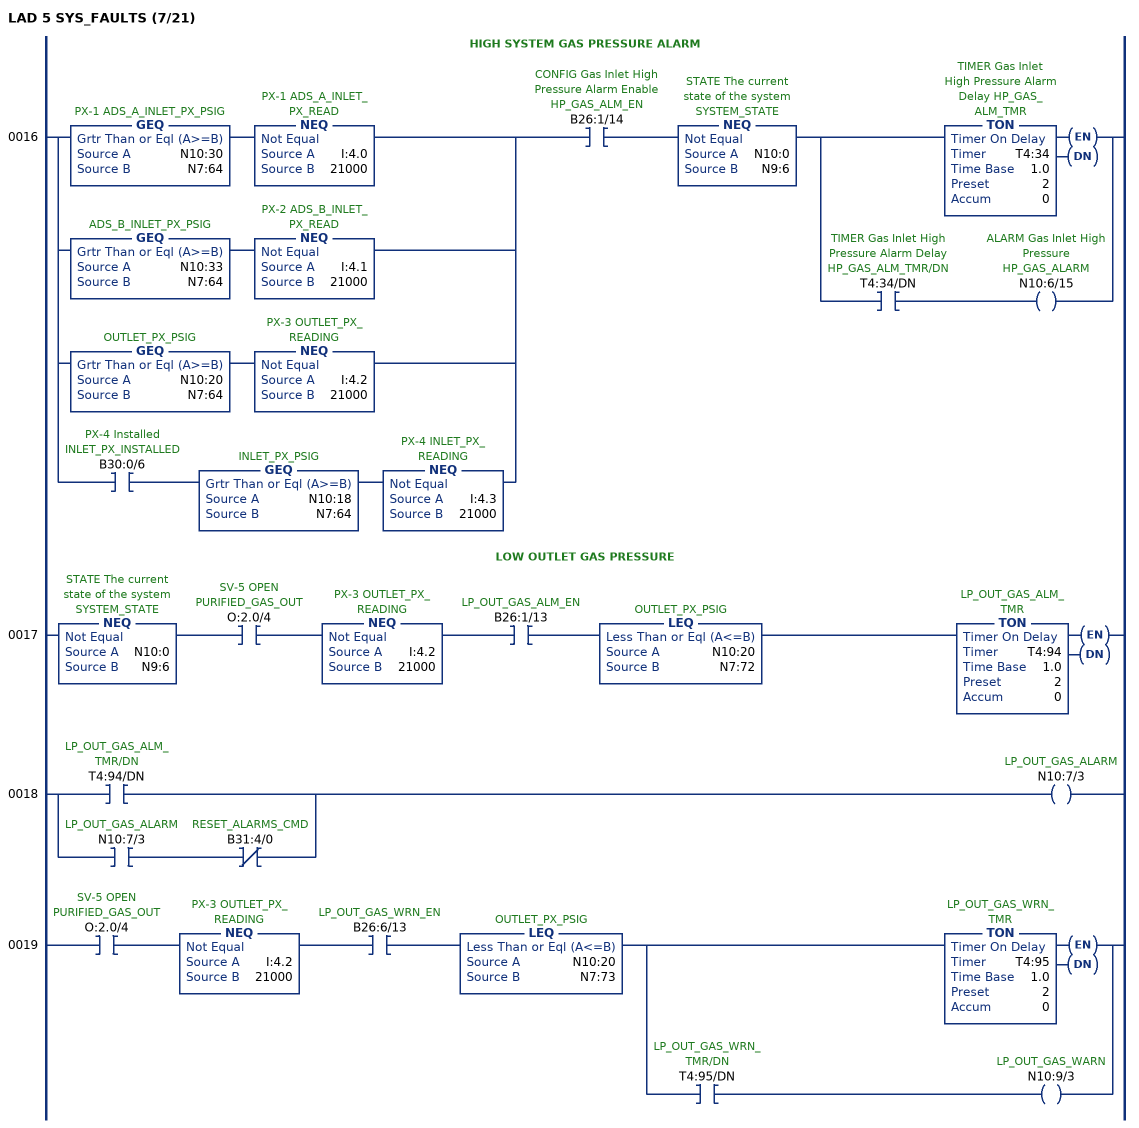
% Rung: 16 %
% TITLE: HIGH SYSTEM GAS PRESSURE ALARM %
SOR BST GEQ N10:30 N7:64 NEQ I:4.0 21000 NXB GEQ N10:33 N7:64 NEQ I:4.1 21000 NXB GEQ N10:20 N7:64 NEQ I:4.2 21000 NXB XIC B30:0/6 GEQ N10:18 N7:64 NEQ I:4.3 21000 BND XIC B26:1/14 NEQ N10:0 N9:6 BST TON T4:34 1.0 2 0 NXB XIC T4:34/DN OTE N10:6/15 BND EOR
%   N10:30  ADS_A_INLET_PX_PSIG  "PX-1" %
%   N7:64  HP_GAS_ALM_SP  "CONFIG Gas Inlet High Pressure Alarm Setpoint" %
%   I:4.0  ADS_A_INLET_PX_READ  "PX-1" %
%   N10:33  ADS_B_INLET_PX_PSIG %
%   I:4.1  ADS_B_INLET_PX_READ  "PX-2" %
%   N10:20  OUTLET_PX_PSIG %
%   I:4.2  OUTLET_PX_READING  "PX-3" %
%   B30:0/6  INLET_PX_INSTALLED  "PX-4 Installed" %
%   N10:18  INLET_PX_PSIG %
%   I:4.3  INLET_PX_READING  "PX-4" %
%   B26:1/14  HP_GAS_ALM_EN  "CONFIG Gas Inlet High Pressure Alarm Enable" %
%   N10:0  SYSTEM_STATE  "STATE The current state of the system" %
%   N9:6  SYSTEM_PURGE %
%   T4:34  HP_GAS_ALM_TMR  "TIMER Gas Inlet High Pressure Alarm Delay" %
%   N10:6/15  HP_GAS_ALARM  "ALARM Gas Inlet High Pressure" %
% Rung: 17 %
% TITLE: LOW OUTLET GAS PRESSURE %
SOR NEQ N10:0 N9:6 XIC O:2.0/4 NEQ I:4.2 21000 XIC B26:1/13 LEQ N10:20 N7:72 TON T4:94 1.0 2 0 EOR
%   N10:0  SYSTEM_STATE  "STATE The current state of the system" %
%   N9:6  SYSTEM_PURGE %
%   O:2.0/4  PURIFIED_GAS_OUT  "SV-5 OPEN" %
%   I:4.2  OUTLET_PX_READING  "PX-3" %
%   B26:1/13  LP_OUT_GAS_ALM_EN %
%   N10:20  OUTLET_PX_PSIG %
%   N7:72  LP_OUT_GAS_ALM_SP %
%   T4:94  LP_OUT_GAS_ALM_TMR %
% Rung: 18 %
SOR BST XIC T4:94/DN NXB XIC N10:7/3 XIO B31:4/0 BND OTE N10:7/3 EOR
%   T4:94  LP_OUT_GAS_ALM_TMR %
%   N10:7/3  LP_OUT_GAS_ALARM %
%   B31:4/0  RESET_ALARMS_CMD %
% Rung: 19 %
SOR XIC O:2.0/4 NEQ I:4.2 21000 XIC B26:6/13 LEQ N10:20 N7:73 BST TON T4:95 1.0 2 0 NXB XIC T4:95/DN OTE N10:9/3 BND EOR
%   O:2.0/4  PURIFIED_GAS_OUT  "SV-5 OPEN" %
%   I:4.2  OUTLET_PX_READING  "PX-3" %
%   B26:6/13  LP_OUT_GAS_WRN_EN %
%   N10:20  OUTLET_PX_PSIG %
%   N7:73  LP_OUT_GAS_WRN_SP %
%   T4:95  LP_OUT_GAS_WRN_TMR %
%   N10:9/3  LP_OUT_GAS_WARN %

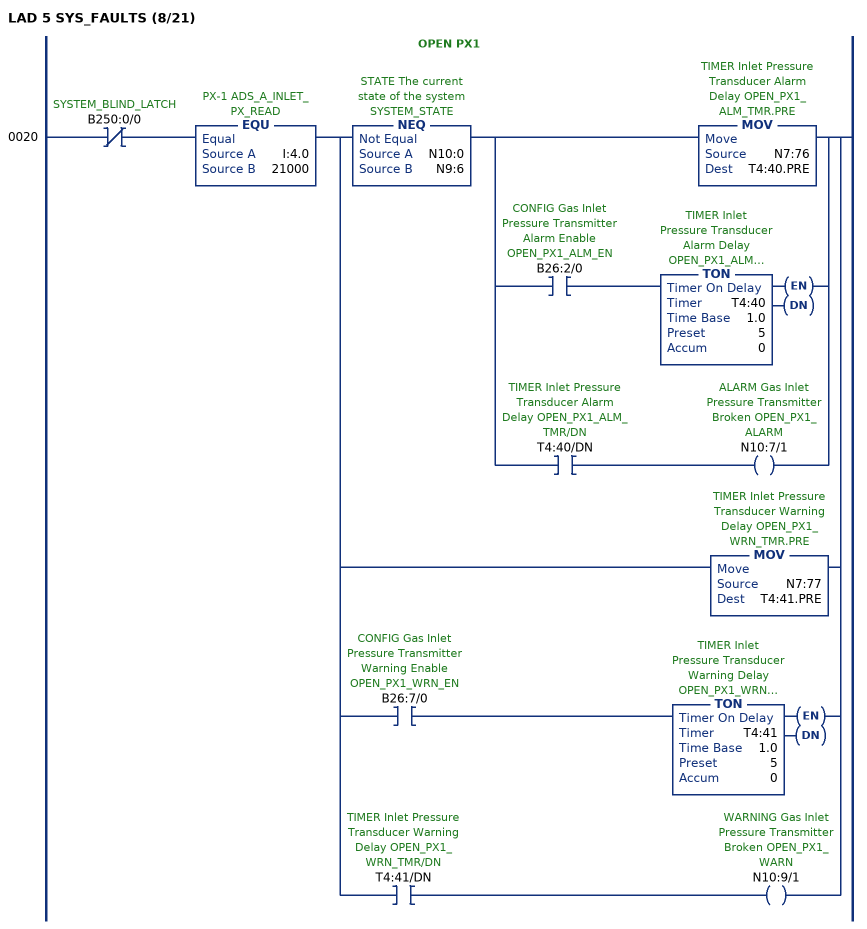
% Rung: 20 %
% TITLE: OPEN PX1 %
SOR XIO B250:0/0 EQU I:4.0 21000 BST NEQ N10:0 N9:6 BST MOV N7:76 T4:40.PRE NXB XIC B26:2/0 TON T4:40 1.0 5 0 NXB XIC T4:40/DN OTE N10:7/1 BND NXB BST MOV N7:77 T4:41.PRE NXB XIC B26:7/0 TON T4:41 1.0 5 0 NXB XIC T4:41/DN OTE N10:9/1 BND BND EOR
%   B250:0/0  SYSTEM_BLIND_LATCH %
%   I:4.0  ADS_A_INLET_PX_READ  "PX-1" %
%   N10:0  SYSTEM_STATE  "STATE The current state of the system" %
%   N9:6  SYSTEM_PURGE %
%   N7:76  OPEN_PX1_ALM_DLY  "CONFIG Gas Inlet Pressure Transducer Alarm Delay" %
%   T4:40  OPEN_PX1_ALM_TMR  "TIMER Inlet Pressure Transducer Alarm Delay" %
%   B26:2/0  OPEN_PX1_ALM_EN  "CONFIG Gas Inlet Pressure Transmitter Alarm Enable" %
%   N10:7/1  OPEN_PX1_ALARM  "ALARM Gas Inlet Pressure Transmitter Broken" %
%   N7:77  OPEN_PX1_WRN_DLY  "CONFIG Gas Inlet Pressure Transducer Warning Delay" %
%   T4:41  OPEN_PX1_WRN_TMR  "TIMER Inlet Pressure Transducer Warning Delay" %
%   B26:7/0  OPEN_PX1_WRN_EN  "CONFIG Gas Inlet Pressure Transmitter Warning Enable" %
%   N10:9/1  OPEN_PX1_WARN  "WARNING Gas Inlet Pressure Transmitter Broken" %

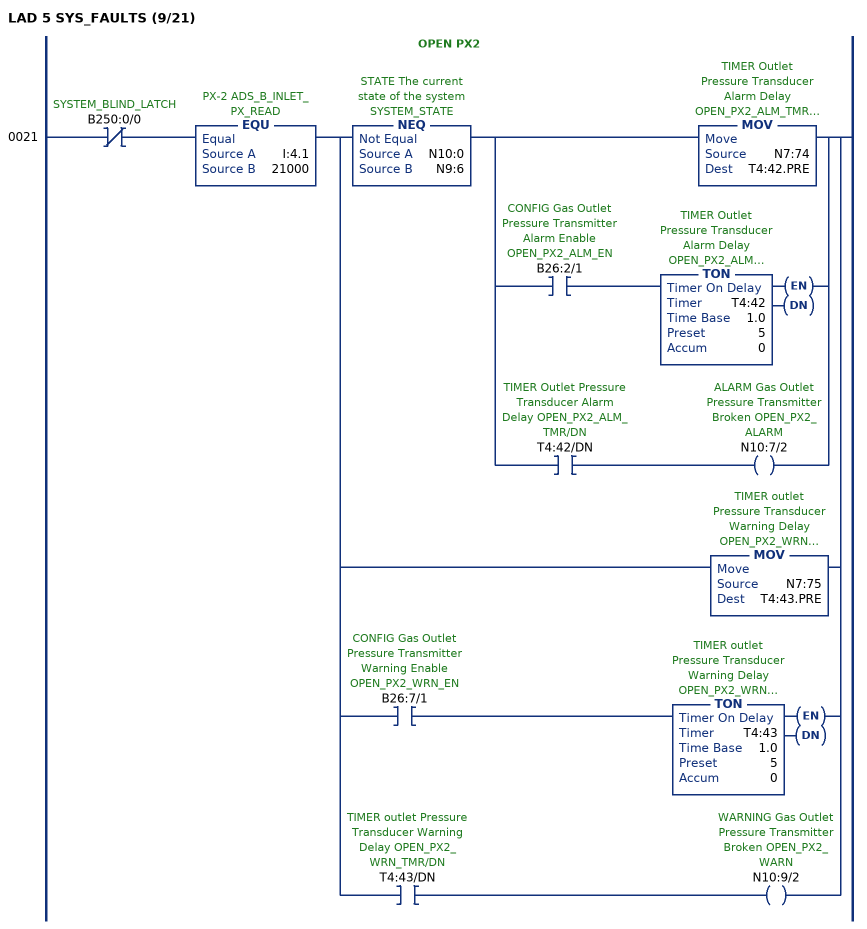
% Rung: 21 %
% TITLE: OPEN PX2 %
SOR XIO B250:0/0 EQU I:4.1 21000 BST NEQ N10:0 N9:6 BST MOV N7:74 T4:42.PRE NXB XIC B26:2/1 TON T4:42 1.0 5 0 NXB XIC T4:42/DN OTE N10:7/2 BND NXB BST MOV N7:75 T4:43.PRE NXB XIC B26:7/1 TON T4:43 1.0 5 0 NXB XIC T4:43/DN OTE N10:9/2 BND BND EOR
%   B250:0/0  SYSTEM_BLIND_LATCH %
%   I:4.1  ADS_B_INLET_PX_READ  "PX-2" %
%   N10:0  SYSTEM_STATE  "STATE The current state of the system" %
%   N9:6  SYSTEM_PURGE %
%   N7:74  OPEN_PX2_ALM_DLY  "CONFIG Gas Outlet Pressure Transducer Alarm Delay" %
%   T4:42  OPEN_PX2_ALM_TMR  "TIMER Outlet Pressure Transducer Alarm Delay" %
%   B26:2/1  OPEN_PX2_ALM_EN  "CONFIG Gas Outlet Pressure Transmitter Alarm Enable" %
%   N10:7/2  OPEN_PX2_ALARM  "ALARM Gas Outlet Pressure Transmitter Broken" %
%   N7:75  OPEN_PX2_WRN_DLY  "CONFIG Gas Outlet Pressure Transducer Warning Delay" %
%   T4:43  OPEN_PX2_WRN_TMR  "TIMER outlet Pressure Transducer Warning Delay" %
%   B26:7/1  OPEN_PX2_WRN_EN  "CONFIG Gas Outlet Pressure Transmitter Warning Enable" %
%   N10:9/2  OPEN_PX2_WARN  "WARNING Gas Outlet Pressure Transmitter Broken" %

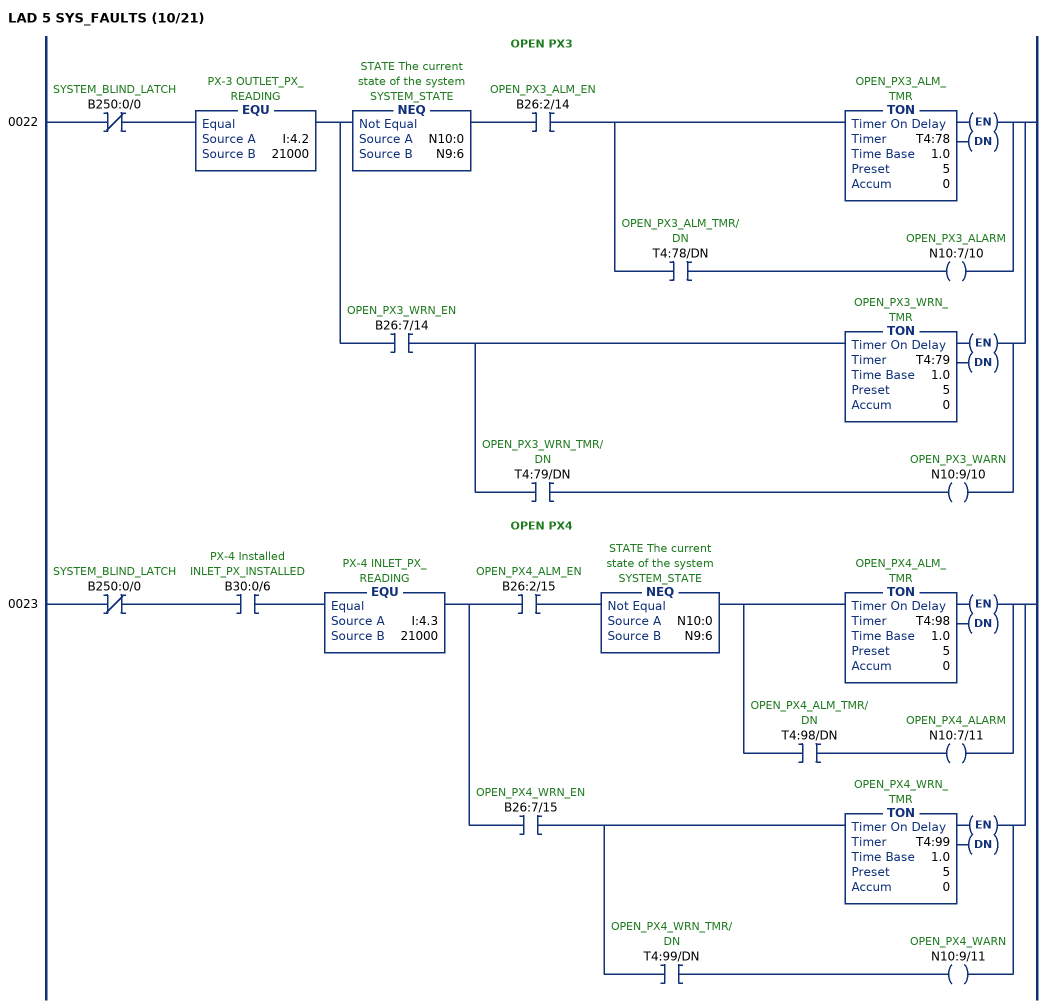
% Rung: 22 %
% TITLE: OPEN PX3 %
SOR XIO B250:0/0 EQU I:4.2 21000 BST NEQ N10:0 N9:6 XIC B26:2/14 BST TON T4:78 1.0 5 0 NXB XIC T4:78/DN OTE N10:7/10 BND NXB XIC B26:7/14 BST TON T4:79 1.0 5 0 NXB XIC T4:79/DN OTE N10:9/10 BND BND EOR
%   B250:0/0  SYSTEM_BLIND_LATCH %
%   I:4.2  OUTLET_PX_READING  "PX-3" %
%   N10:0  SYSTEM_STATE  "STATE The current state of the system" %
%   N9:6  SYSTEM_PURGE %
%   B26:2/14  OPEN_PX3_ALM_EN %
%   T4:78  OPEN_PX3_ALM_TMR %
%   N10:7/10  OPEN_PX3_ALARM %
%   B26:7/14  OPEN_PX3_WRN_EN %
%   T4:79  OPEN_PX3_WRN_TMR %
%   N10:9/10  OPEN_PX3_WARN %
% Rung: 23 %
% TITLE: OPEN PX4 %
SOR XIO B250:0/0 XIC B30:0/6 EQU I:4.3 21000 BST XIC B26:2/15 NEQ N10:0 N9:6 BST TON T4:98 1.0 5 0 NXB XIC T4:98/DN OTE N10:7/11 BND NXB XIC B26:7/15 BST TON T4:99 1.0 5 0 NXB XIC T4:99/DN OTE N10:9/11 BND BND EOR
%   B250:0/0  SYSTEM_BLIND_LATCH %
%   B30:0/6  INLET_PX_INSTALLED  "PX-4 Installed" %
%   I:4.3  INLET_PX_READING  "PX-4" %
%   B26:2/15  OPEN_PX4_ALM_EN %
%   N10:0  SYSTEM_STATE  "STATE The current state of the system" %
%   N9:6  SYSTEM_PURGE %
%   T4:98  OPEN_PX4_ALM_TMR %
%   N10:7/11  OPEN_PX4_ALARM %
%   B26:7/15  OPEN_PX4_WRN_EN %
%   T4:99  OPEN_PX4_WRN_TMR %
%   N10:9/11  OPEN_PX4_WARN %

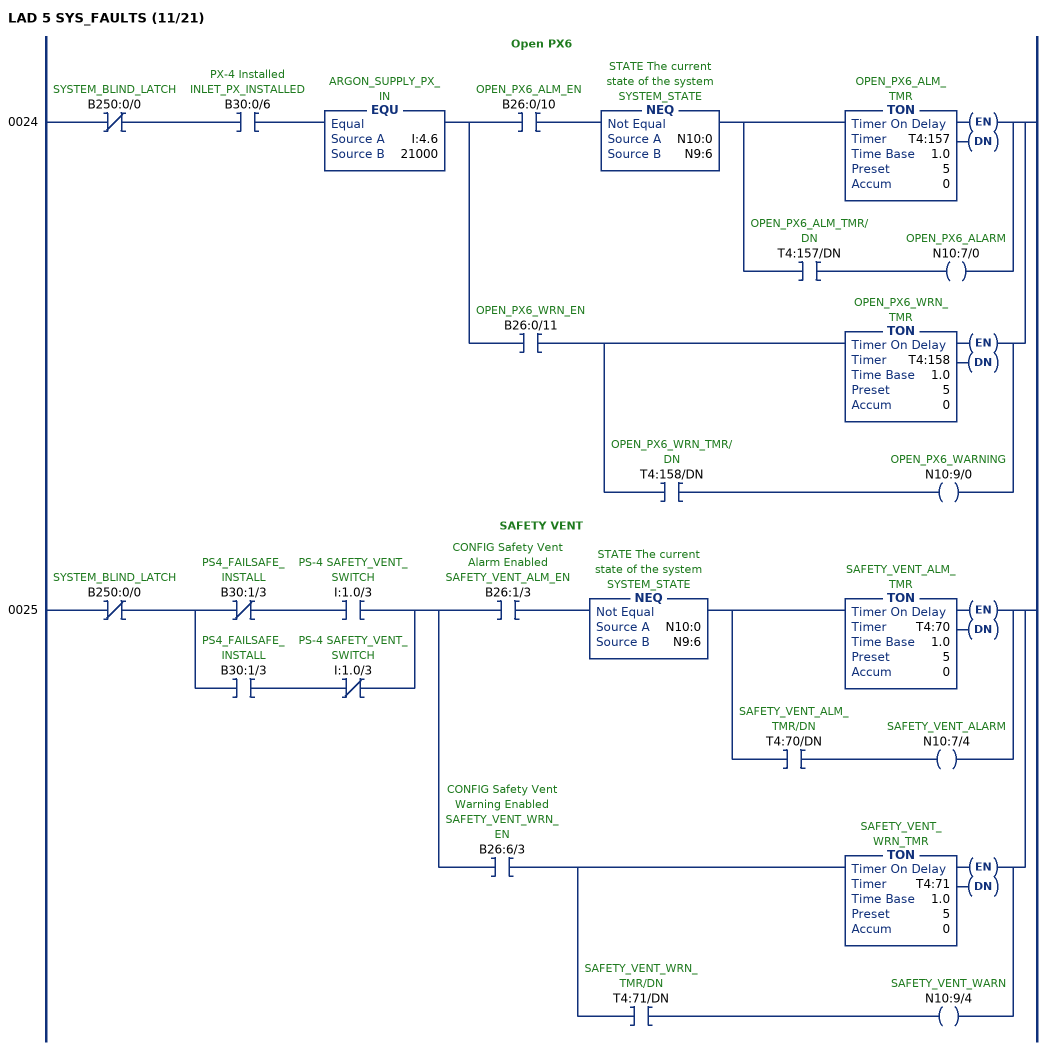
% Rung: 24 %
% TITLE: Open PX6 %
SOR XIO B250:0/0 XIC B30:0/6 EQU I:4.6 21000 BST XIC B26:0/10 NEQ N10:0 N9:6 BST TON T4:157 1.0 5 0 NXB XIC T4:157/DN OTE N10:7/0 BND NXB XIC B26:0/11 BST TON T4:158 1.0 5 0 NXB XIC T4:158/DN OTE N10:9/0 BND BND EOR
%   B250:0/0  SYSTEM_BLIND_LATCH %
%   B30:0/6  INLET_PX_INSTALLED  "PX-4 Installed" %
%   I:4.6  ARGON_SUPPLY_PX_IN %
%   B26:0/10  OPEN_PX6_ALM_EN %
%   N10:0  SYSTEM_STATE  "STATE The current state of the system" %
%   N9:6  SYSTEM_PURGE %
%   T4:157  OPEN_PX6_ALM_TMR %
%   N10:7/0  OPEN_PX6_ALARM %
%   B26:0/11  OPEN_PX6_WRN_EN %
%   T4:158  OPEN_PX6_WRN_TMR %
%   N10:9/0  OPEN_PX6_WARNING %
% Rung: 25 %
% TITLE: SAFETY VENT %
SOR XIO B250:0/0 BST XIO B30:1/3 XIC I:1.0/3 NXB XIC B30:1/3 XIO I:1.0/3 BND BST XIC B26:1/3 NEQ N10:0 N9:6 BST TON T4:70 1.0 5 0 NXB XIC T4:70/DN OTE N10:7/4 BND NXB XIC B26:6/3 BST TON T4:71 1.0 5 0 NXB XIC T4:71/DN OTE N10:9/4 BND BND EOR
%   B250:0/0  SYSTEM_BLIND_LATCH %
%   B30:1/3  PS4_FAILSAFE_INSTALL %
%   I:1.0/3  SAFETY_VENT_SWITCH  "PS-4" %
%   B26:1/3  SAFETY_VENT_ALM_EN  "CONFIG Safety Vent Alarm Enabled" %
%   N10:0  SYSTEM_STATE  "STATE The current state of the system" %
%   N9:6  SYSTEM_PURGE %
%   T4:70  SAFETY_VENT_ALM_TMR %
%   N10:7/4  SAFETY_VENT_ALARM %
%   B26:6/3  SAFETY_VENT_WRN_EN  "CONFIG Safety Vent Warning Enabled" %
%   T4:71  SAFETY_VENT_WRN_TMR %
%   N10:9/4  SAFETY_VENT_WARN %

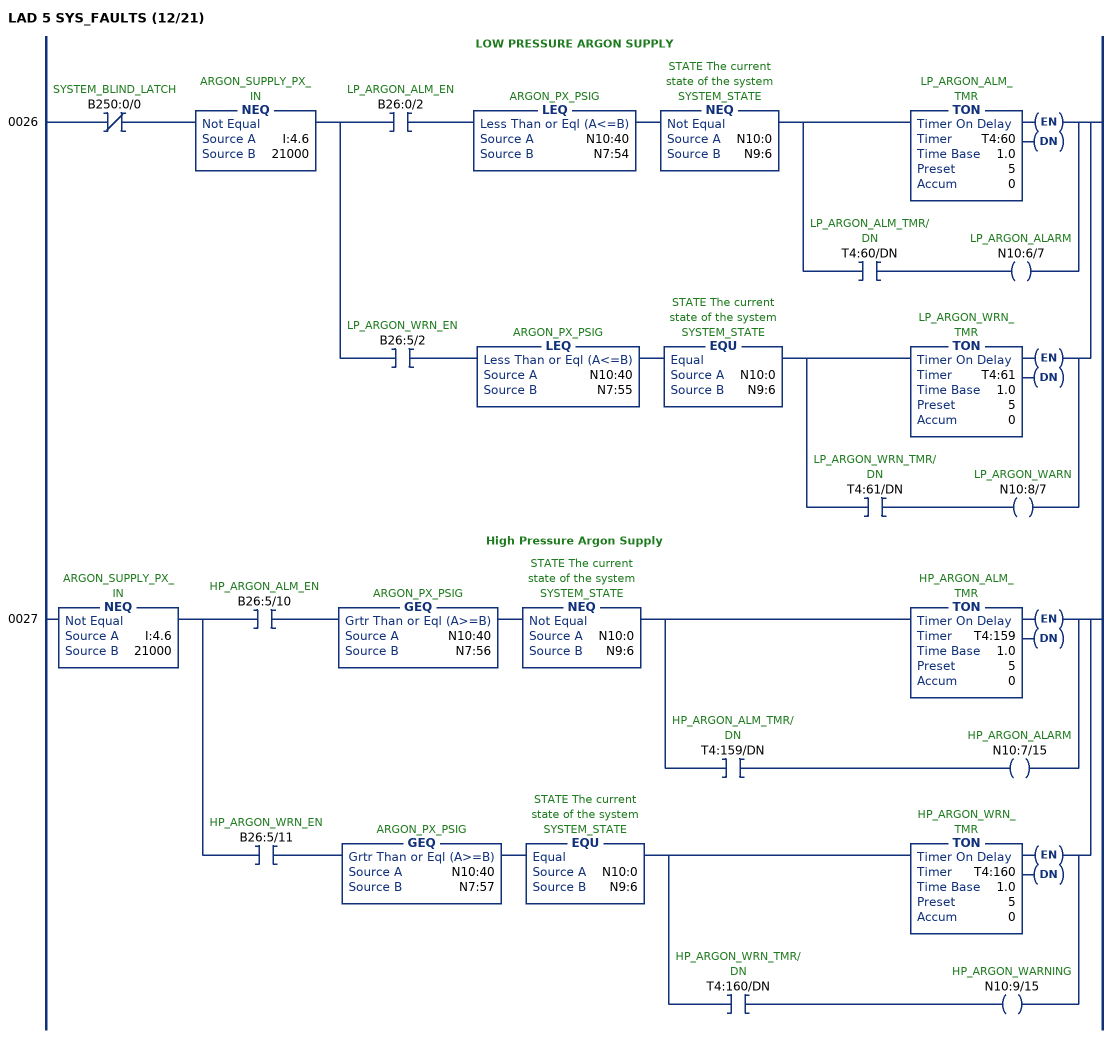
% Rung: 26 %
% TITLE: LOW PRESSURE ARGON SUPPLY %
SOR XIO B250:0/0 NEQ I:4.6 21000 BST XIC B26:0/2 LEQ N10:40 N7:54 NEQ N10:0 N9:6 BST TON T4:60 1.0 5 0 NXB XIC T4:60/DN OTE N10:6/7 BND NXB XIC B26:5/2 LEQ N10:40 N7:55 EQU N10:0 N9:6 BST TON T4:61 1.0 5 0 NXB XIC T4:61/DN OTE N10:8/7 BND BND EOR
%   B250:0/0  SYSTEM_BLIND_LATCH %
%   I:4.6  ARGON_SUPPLY_PX_IN %
%   B26:0/2  LP_ARGON_ALM_EN %
%   N10:40  ARGON_PX_PSIG %
%   N7:54  LP_ARGON_ALM_SP %
%   N10:0  SYSTEM_STATE  "STATE The current state of the system" %
%   N9:6  SYSTEM_PURGE %
%   T4:60  LP_ARGON_ALM_TMR %
%   N10:6/7  LP_ARGON_ALARM %
%   B26:5/2  LP_ARGON_WRN_EN %
%   N7:55  LP_ARGON_WRN_SP %
%   T4:61  LP_ARGON_WRN_TMR %
%   N10:8/7  LP_ARGON_WARN %
% Rung: 27 %
% TITLE: High Pressure Argon Supply %
SOR NEQ I:4.6 21000 BST XIC B26:5/10 GEQ N10:40 N7:56 NEQ N10:0 N9:6 BST TON T4:159 1.0 5 0 NXB XIC T4:159/DN OTE N10:7/15 BND NXB XIC B26:5/11 GEQ N10:40 N7:57 EQU N10:0 N9:6 BST TON T4:160 1.0 5 0 NXB XIC T4:160/DN OTE N10:9/15 BND BND EOR
%   I:4.6  ARGON_SUPPLY_PX_IN %
%   B26:5/10  HP_ARGON_ALM_EN %
%   N10:40  ARGON_PX_PSIG %
%   N7:56  HP_ARGON_ALM_SP %
%   N10:0  SYSTEM_STATE  "STATE The current state of the system" %
%   N9:6  SYSTEM_PURGE %
%   T4:159  HP_ARGON_ALM_TMR %
%   N10:7/15  HP_ARGON_ALARM %
%   B26:5/11  HP_ARGON_WRN_EN %
%   N7:57  HP_ARGON_WRN_SP %
%   T4:160  HP_ARGON_WRN_TMR %
%   N10:9/15  HP_ARGON_WARNING %

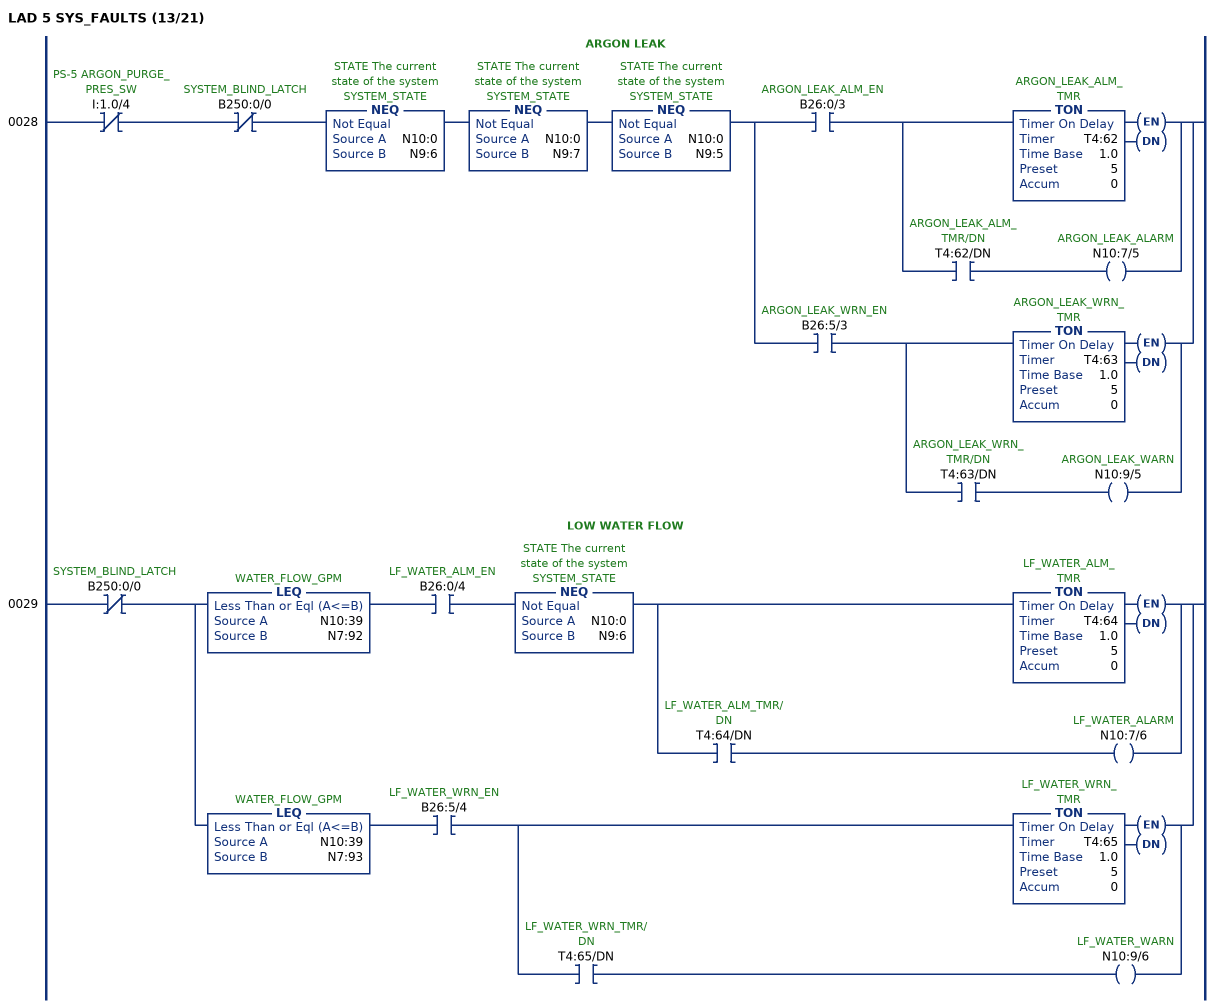
% Rung: 28 %
% TITLE: ARGON LEAK %
SOR XIO I:1.0/4 XIO B250:0/0 NEQ N10:0 N9:6 NEQ N10:0 N9:7 NEQ N10:0 N9:5 BST XIC B26:0/3 BST TON T4:62 1.0 5 0 NXB XIC T4:62/DN OTE N10:7/5 BND NXB XIC B26:5/3 BST TON T4:63 1.0 5 0 NXB XIC T4:63/DN OTE N10:9/5 BND BND EOR
%   I:1.0/4  ARGON_PURGE_PRES_SW  "PS-5" %
%   B250:0/0  SYSTEM_BLIND_LATCH %
%   N10:0  SYSTEM_STATE  "STATE The current state of the system" %
%   N9:6  SYSTEM_PURGE %
%   N9:7  SYSTEM_COLD_START %
%   N9:5  SYSTEM_QUICK_START %
%   B26:0/3  ARGON_LEAK_ALM_EN %
%   T4:62  ARGON_LEAK_ALM_TMR %
%   N10:7/5  ARGON_LEAK_ALARM %
%   B26:5/3  ARGON_LEAK_WRN_EN %
%   T4:63  ARGON_LEAK_WRN_TMR %
%   N10:9/5  ARGON_LEAK_WARN %
% Rung: 29 %
% TITLE: LOW WATER FLOW %
SOR XIO B250:0/0 BST LEQ N10:39 N7:92 XIC B26:0/4 NEQ N10:0 N9:6 BST TON T4:64 1.0 5 0 NXB XIC T4:64/DN OTE N10:7/6 BND NXB LEQ N10:39 N7:93 XIC B26:5/4 BST TON T4:65 1.0 5 0 NXB XIC T4:65/DN OTE N10:9/6 BND BND EOR
%   B250:0/0  SYSTEM_BLIND_LATCH %
%   N10:39  WATER_FLOW_GPM %
%   N7:92  LF_WATER_ALM_SP %
%   B26:0/4  LF_WATER_ALM_EN %
%   N10:0  SYSTEM_STATE  "STATE The current state of the system" %
%   N9:6  SYSTEM_PURGE %
%   T4:64  LF_WATER_ALM_TMR %
%   N10:7/6  LF_WATER_ALARM %
%   N7:93  LF_WATER_WRN_SP %
%   B26:5/4  LF_WATER_WRN_EN %
%   T4:65  LF_WATER_WRN_TMR %
%   N10:9/6  LF_WATER_WARN %

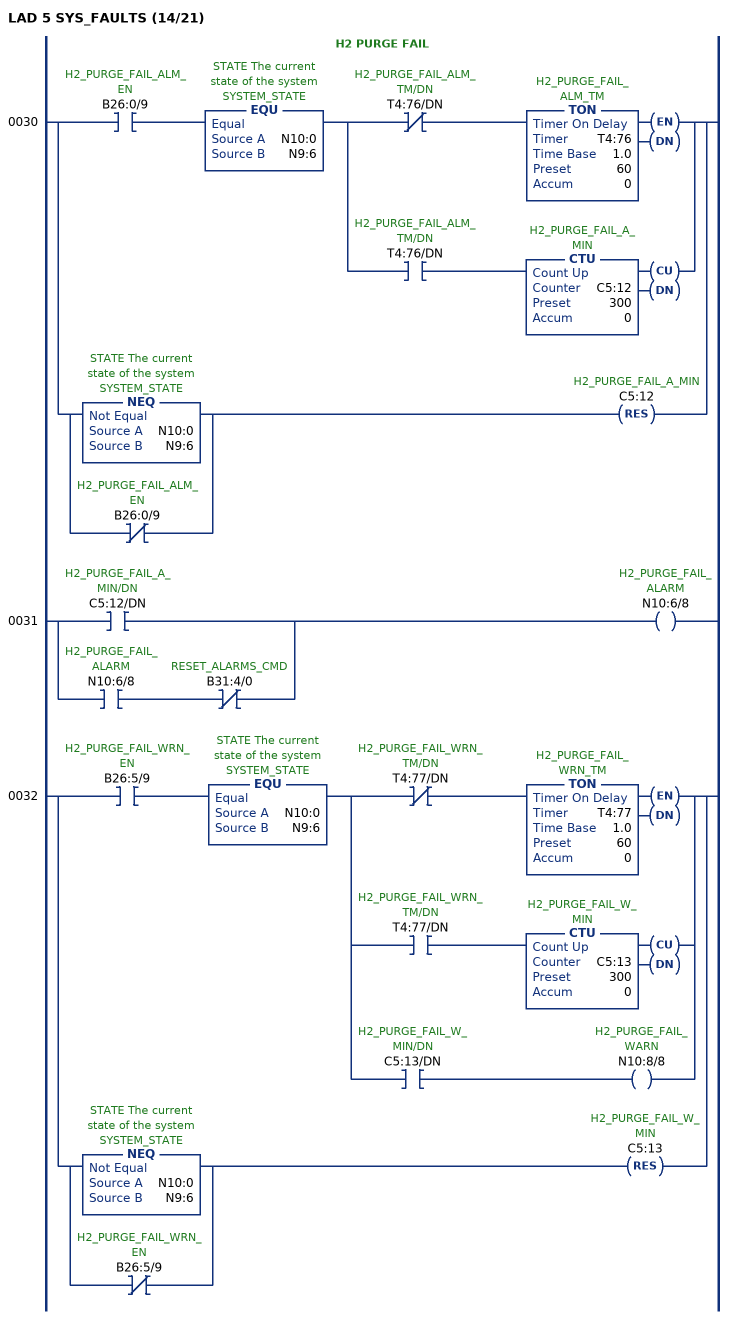
% Rung: 30 %
% TITLE: H2 PURGE FAIL %
SOR BST XIC B26:0/9 EQU N10:0 N9:6 BST XIO T4:76/DN TON T4:76 1.0 60 0 NXB XIC T4:76/DN CTU C5:12 300 0 BND NXB BST NEQ N10:0 N9:6 NXB XIO B26:0/9 BND RES C5:12 BND EOR
%   B26:0/9  H2_PURGE_FAIL_ALM_EN %
%   N10:0  SYSTEM_STATE  "STATE The current state of the system" %
%   N9:6  SYSTEM_PURGE %
%   T4:76  H2_PURGE_FAIL_ALM_TM %
%   C5:12  H2_PURGE_FAIL_A_MIN %
% Rung: 31 %
SOR BST XIC C5:12/DN NXB XIC N10:6/8 XIO B31:4/0 BND OTE N10:6/8 EOR
%   C5:12  H2_PURGE_FAIL_A_MIN %
%   N10:6/8  H2_PURGE_FAIL_ALARM %
%   B31:4/0  RESET_ALARMS_CMD %
% Rung: 32 %
SOR BST XIC B26:5/9 EQU N10:0 N9:6 BST XIO T4:77/DN TON T4:77 1.0 60 0 NXB XIC T4:77/DN CTU C5:13 300 0 NXB XIC C5:13/DN OTE N10:8/8 BND NXB BST NEQ N10:0 N9:6 NXB XIO B26:5/9 BND RES C5:13 BND EOR
%   B26:5/9  H2_PURGE_FAIL_WRN_EN %
%   N10:0  SYSTEM_STATE  "STATE The current state of the system" %
%   N9:6  SYSTEM_PURGE %
%   T4:77  H2_PURGE_FAIL_WRN_TM %
%   C5:13  H2_PURGE_FAIL_W_MIN %
%   N10:8/8  H2_PURGE_FAIL_WARN %

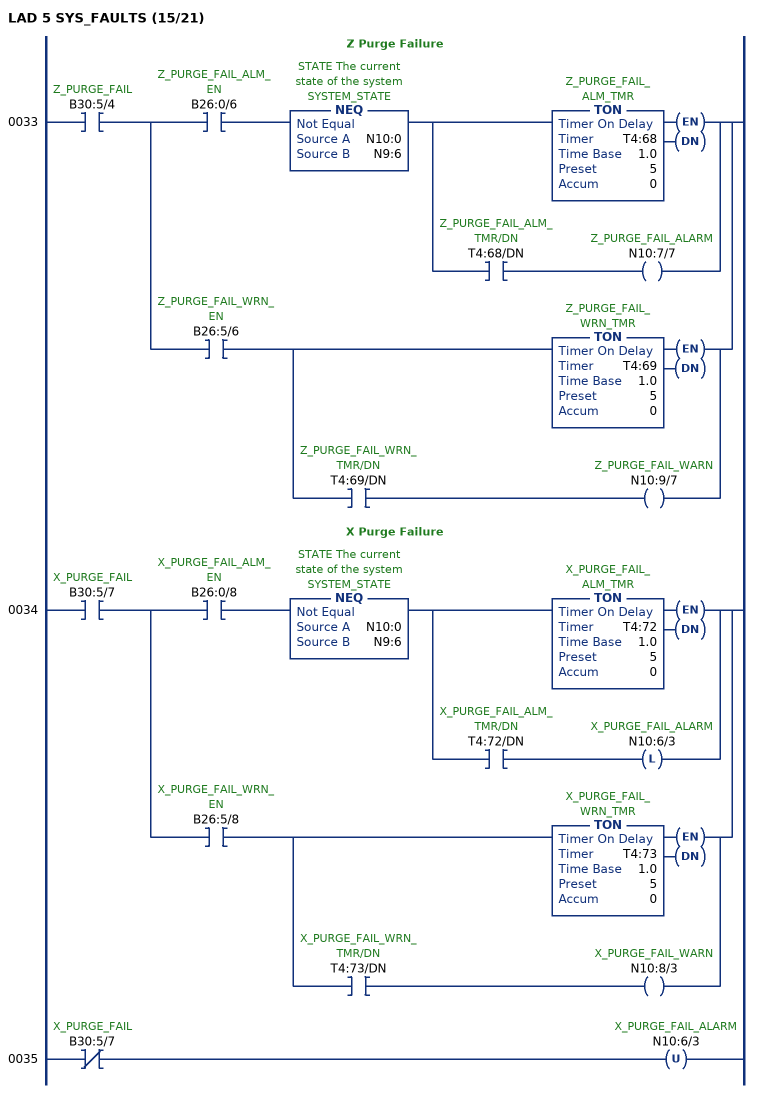
% Rung: 33 %
% TITLE: Z Purge Failure %
SOR XIC B30:5/4 BST XIC B26:0/6 NEQ N10:0 N9:6 BST TON T4:68 1.0 5 0 NXB XIC T4:68/DN OTE N10:7/7 BND NXB XIC B26:5/6 BST TON T4:69 1.0 5 0 NXB XIC T4:69/DN OTE N10:9/7 BND BND EOR
%   B30:5/4  Z_PURGE_FAIL %
%   B26:0/6  Z_PURGE_FAIL_ALM_EN %
%   N10:0  SYSTEM_STATE  "STATE The current state of the system" %
%   N9:6  SYSTEM_PURGE %
%   T4:68  Z_PURGE_FAIL_ALM_TMR %
%   N10:7/7  Z_PURGE_FAIL_ALARM %
%   B26:5/6  Z_PURGE_FAIL_WRN_EN %
%   T4:69  Z_PURGE_FAIL_WRN_TMR %
%   N10:9/7  Z_PURGE_FAIL_WARN %
% Rung: 34 %
% TITLE: X Purge Failure %
SOR XIC B30:5/7 BST XIC B26:0/8 NEQ N10:0 N9:6 BST TON T4:72 1.0 5 0 NXB XIC T4:72/DN OTL N10:6/3 BND NXB XIC B26:5/8 BST TON T4:73 1.0 5 0 NXB XIC T4:73/DN OTE N10:8/3 BND BND EOR
%   B30:5/7  X_PURGE_FAIL %
%   B26:0/8  X_PURGE_FAIL_ALM_EN %
%   N10:0  SYSTEM_STATE  "STATE The current state of the system" %
%   N9:6  SYSTEM_PURGE %
%   T4:72  X_PURGE_FAIL_ALM_TMR %
%   N10:6/3  X_PURGE_FAIL_ALARM %
%   B26:5/8  X_PURGE_FAIL_WRN_EN %
%   T4:73  X_PURGE_FAIL_WRN_TMR %
%   N10:8/3  X_PURGE_FAIL_WARN %
% Rung: 35 %
SOR XIO B30:5/7 OTU N10:6/3 EOR
%   B30:5/7  X_PURGE_FAIL %
%   N10:6/3  X_PURGE_FAIL_ALARM %

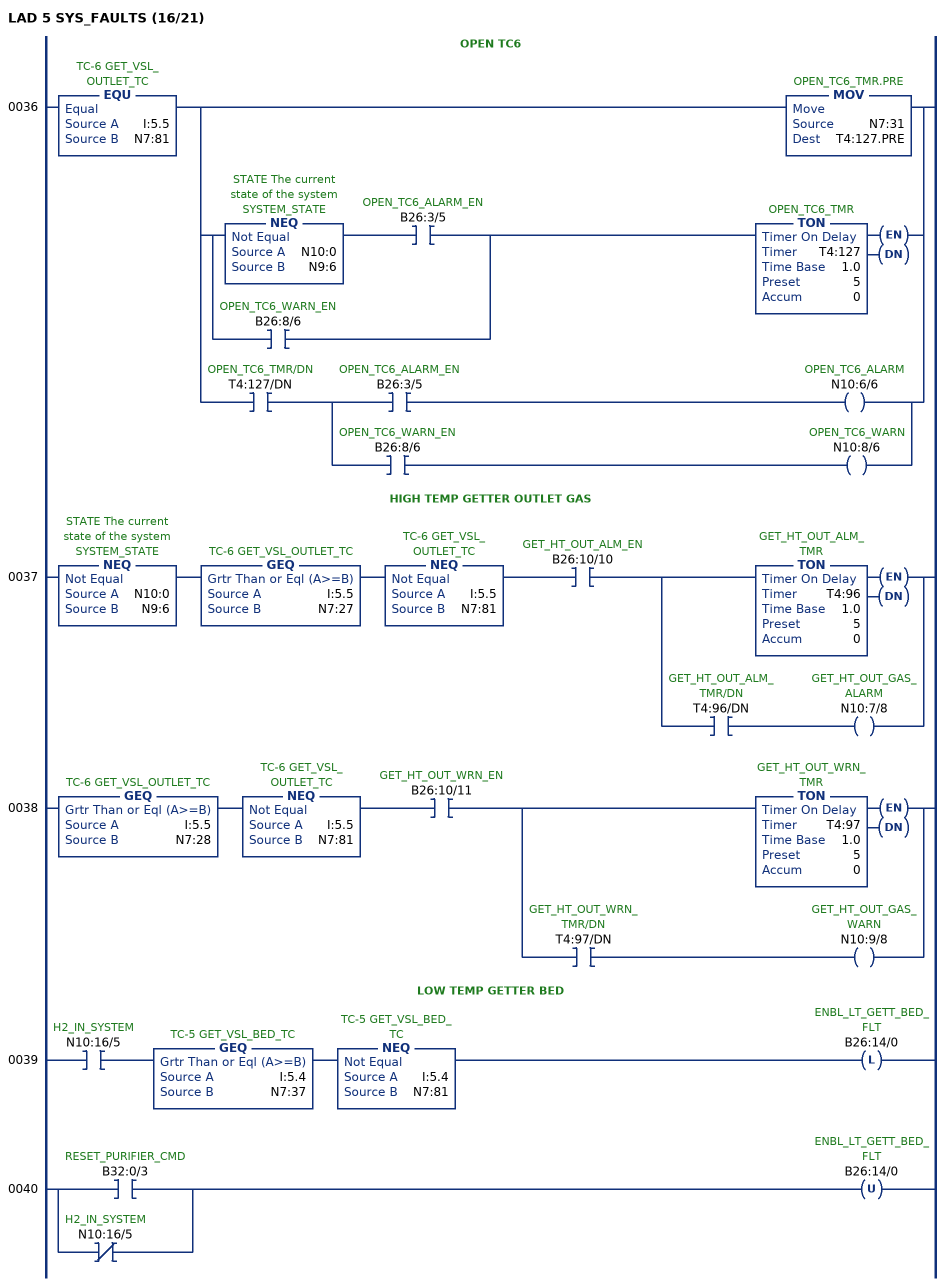
% Rung: 36 %
% TITLE: OPEN TC6 %
SOR EQU I:5.5 N7:81 BST MOV N7:31 T4:127.PRE NXB BST NEQ N10:0 N9:6 XIC B26:3/5 NXB XIC B26:8/6 BND TON T4:127 1.0 5 0 NXB XIC T4:127/DN BST XIC B26:3/5 OTE N10:6/6 NXB XIC B26:8/6 OTE N10:8/6 BND BND EOR
%   I:5.5  GET_VSL_OUTLET_TC  "TC-6" %
%   N7:81  TC_OPEN_SP  "CONFIG The value read by an open TC input" %
%   N7:31  OPEN_TC_DLY %
%   T4:127  OPEN_TC6_TMR %
%   N10:0  SYSTEM_STATE  "STATE The current state of the system" %
%   N9:6  SYSTEM_PURGE %
%   B26:3/5  OPEN_TC6_ALARM_EN %
%   B26:8/6  OPEN_TC6_WARN_EN %
%   N10:6/6  OPEN_TC6_ALARM %
%   N10:8/6  OPEN_TC6_WARN %
% Rung: 37 %
% TITLE: HIGH TEMP GETTER OUTLET GAS %
SOR NEQ N10:0 N9:6 GEQ I:5.5 N7:27 NEQ I:5.5 N7:81 XIC B26:10/10 BST TON T4:96 1.0 5 0 NXB XIC T4:96/DN OTE N10:7/8 BND EOR
%   N10:0  SYSTEM_STATE  "STATE The current state of the system" %
%   N9:6  SYSTEM_PURGE %
%   I:5.5  GET_VSL_OUTLET_TC  "TC-6" %
%   N7:27  GET_HT_OUT_ALM_SP %
%   N7:81  TC_OPEN_SP  "CONFIG The value read by an open TC input" %
%   B26:10/10  GET_HT_OUT_ALM_EN %
%   T4:96  GET_HT_OUT_ALM_TMR %
%   N10:7/8  GET_HT_OUT_GAS_ALARM %
% Rung: 38 %
SOR GEQ I:5.5 N7:28 NEQ I:5.5 N7:81 XIC B26:10/11 BST TON T4:97 1.0 5 0 NXB XIC T4:97/DN OTE N10:9/8 BND EOR
%   I:5.5  GET_VSL_OUTLET_TC  "TC-6" %
%   N7:28  GET_HT_OUT_WRN_SP %
%   N7:81  TC_OPEN_SP  "CONFIG The value read by an open TC input" %
%   B26:10/11  GET_HT_OUT_WRN_EN %
%   T4:97  GET_HT_OUT_WRN_TMR %
%   N10:9/8  GET_HT_OUT_GAS_WARN %
% Rung: 39 %
% TITLE: LOW TEMP GETTER BED %
SOR XIC N10:16/5 GEQ I:5.4 N7:37 NEQ I:5.4 N7:81 OTL B26:14/0 EOR
%   N10:16/5  H2_IN_SYSTEM %
%   I:5.4  GET_VSL_BED_TC  "TC-5" %
%   N7:37  GET_LT_SHUTDOWN_SP %
%   N7:81  TC_OPEN_SP  "CONFIG The value read by an open TC input" %
%   B26:14/0  ENBL_LT_GETT_BED_FLT %
% Rung: 40 %
SOR BST XIC B32:0/3 NXB XIO N10:16/5 BND OTU B26:14/0 EOR
%   B32:0/3  RESET_PURIFIER_CMD %
%   N10:16/5  H2_IN_SYSTEM %
%   B26:14/0  ENBL_LT_GETT_BED_FLT %

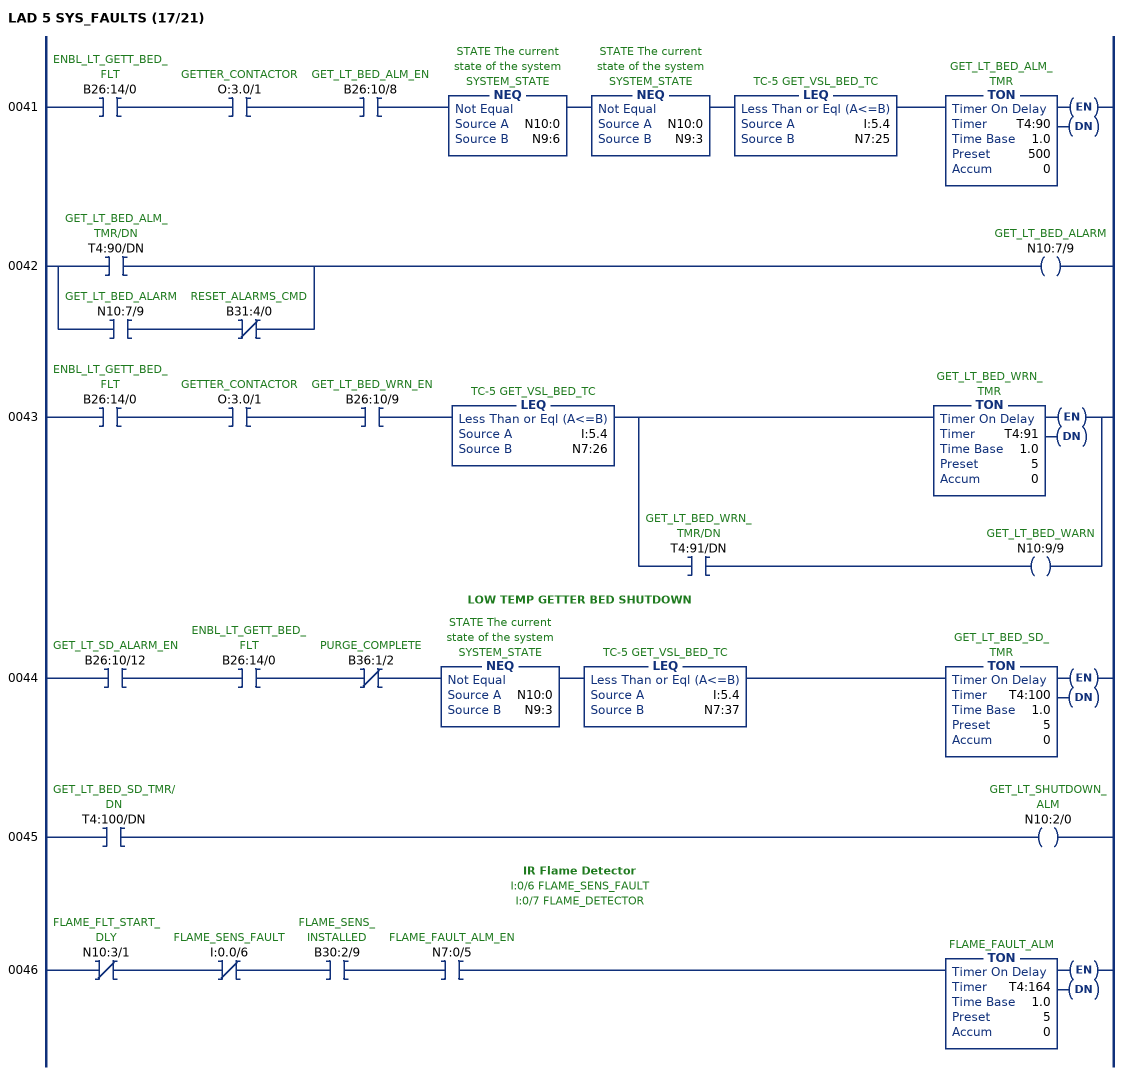
% Rung: 41 %
SOR XIC B26:14/0 XIC O:3.0/1 XIC B26:10/8 NEQ N10:0 N9:6 NEQ N10:0 N9:3 LEQ I:5.4 N7:25 TON T4:90 1.0 500 0 EOR
%   B26:14/0  ENBL_LT_GETT_BED_FLT %
%   O:3.0/1  GETTER_CONTACTOR %
%   B26:10/8  GET_LT_BED_ALM_EN %
%   N10:0  SYSTEM_STATE  "STATE The current state of the system" %
%   N9:6  SYSTEM_PURGE %
%   N9:3  SYSTEM_MANUAL  "STATE System Manual" %
%   I:5.4  GET_VSL_BED_TC  "TC-5" %
%   N7:25  GET_LT_BED_ALM_SP %
%   T4:90  GET_LT_BED_ALM_TMR %
% Rung: 42 %
SOR BST XIC T4:90/DN NXB XIC N10:7/9 XIO B31:4/0 BND OTE N10:7/9 EOR
%   T4:90  GET_LT_BED_ALM_TMR %
%   N10:7/9  GET_LT_BED_ALARM %
%   B31:4/0  RESET_ALARMS_CMD %
% Rung: 43 %
SOR XIC B26:14/0 XIC O:3.0/1 XIC B26:10/9 LEQ I:5.4 N7:26 BST TON T4:91 1.0 5 0 NXB XIC T4:91/DN OTE N10:9/9 BND EOR
%   B26:14/0  ENBL_LT_GETT_BED_FLT %
%   O:3.0/1  GETTER_CONTACTOR %
%   B26:10/9  GET_LT_BED_WRN_EN %
%   I:5.4  GET_VSL_BED_TC  "TC-5" %
%   N7:26  GET_LT_BED_WRN_SP %
%   T4:91  GET_LT_BED_WRN_TMR %
%   N10:9/9  GET_LT_BED_WARN %
% Rung: 44 %
% TITLE: LOW TEMP GETTER BED SHUTDOWN %
SOR XIC B26:10/12 XIC B26:14/0 XIO B36:1/2 NEQ N10:0 N9:3 LEQ I:5.4 N7:37 TON T4:100 1.0 5 0 EOR
%   B26:10/12  GET_LT_SD_ALARM_EN %
%   B26:14/0  ENBL_LT_GETT_BED_FLT %
%   B36:1/2  PURGE_COMPLETE %
%   N10:0  SYSTEM_STATE  "STATE The current state of the system" %
%   N9:3  SYSTEM_MANUAL  "STATE System Manual" %
%   I:5.4  GET_VSL_BED_TC  "TC-5" %
%   N7:37  GET_LT_SHUTDOWN_SP %
%   T4:100  GET_LT_BED_SD_TMR %
% Rung: 45 %
SOR XIC T4:100/DN OTE N10:2/0 EOR
%   T4:100  GET_LT_BED_SD_TMR %
%   N10:2/0  GET_LT_SHUTDOWN_ALM %
% Rung: 46 %
% TITLE: IR Flame Detector %
% I:0/6 FLAME_SENS_FAULT
% I:0/7 FLAME_DETECTOR %
SOR XIO N10:3/1 XIO I:0.0/6 XIC B30:2/9 XIC N7:0/5 TON T4:164 1.0 5 0 EOR
%   N10:3/1  FLAME_FLT_START_DLY %
%   I:0.0/6  FLAME_SENS_FAULT %
%   B30:2/9  FLAME_SENS_INSTALLED %
%   N7:0/5  FLAME_FAULT_ALM_EN %
%   T4:164  FLAME_FAULT_ALM %

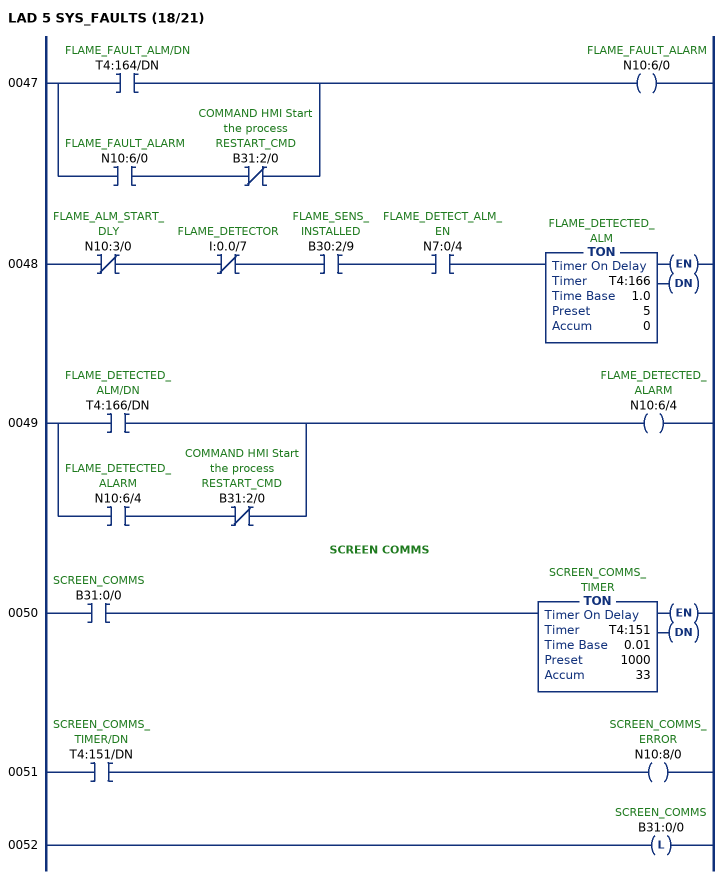
% Rung: 47 %
SOR BST XIC T4:164/DN NXB XIC N10:6/0 XIO B31:2/0 BND OTE N10:6/0 EOR
%   T4:164  FLAME_FAULT_ALM %
%   N10:6/0  FLAME_FAULT_ALARM %
%   B31:2/0  RESTART_CMD  "COMMAND HMI Start the process" %
% Rung: 48 %
SOR XIO N10:3/0 XIO I:0.0/7 XIC B30:2/9 XIC N7:0/4 TON T4:166 1.0 5 0 EOR
%   N10:3/0  FLAME_ALM_START_DLY %
%   I:0.0/7  FLAME_DETECTOR %
%   B30:2/9  FLAME_SENS_INSTALLED %
%   N7:0/4  FLAME_DETECT_ALM_EN %
%   T4:166  FLAME_DETECTED_ALM %
% Rung: 49 %
SOR BST XIC T4:166/DN NXB XIC N10:6/4 XIO B31:2/0 BND OTE N10:6/4 EOR
%   T4:166  FLAME_DETECTED_ALM %
%   N10:6/4  FLAME_DETECTED_ALARM %
%   B31:2/0  RESTART_CMD  "COMMAND HMI Start the process" %
% Rung: 50 %
% TITLE: SCREEN COMMS %
SOR XIC B31:0/0 TON T4:151 0.01 1000 33 EOR
%   B31:0/0  SCREEN_COMMS %
%   T4:151  SCREEN_COMMS_TIMER %
% Rung: 51 %
SOR XIC T4:151/DN OTE N10:8/0 EOR
%   T4:151  SCREEN_COMMS_TIMER %
%   N10:8/0  SCREEN_COMMS_ERROR %
% Rung: 52 %
SOR OTL B31:0/0 EOR
%   B31:0/0  SCREEN_COMMS %

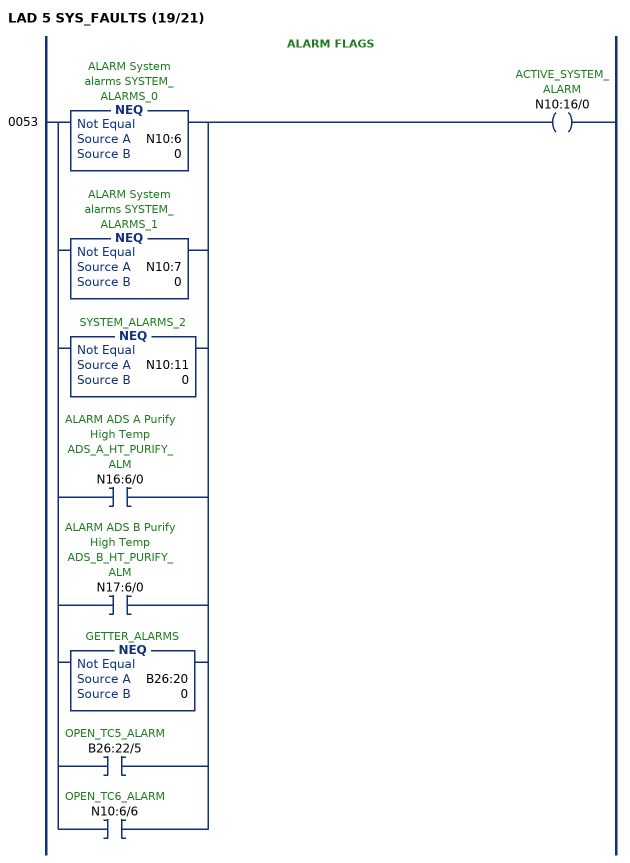
% Rung: 53 %
% TITLE: ALARM FLAGS %
SOR BST NEQ N10:6 0 NXB NEQ N10:7 0 NXB NEQ N10:11 0 NXB XIC N16:6/0 NXB XIC N17:6/0 NXB NEQ B26:20 0 NXB XIC B26:22/5 NXB XIC N10:6/6 BND OTE N10:16/0 EOR
%   N10:6  SYSTEM_ALARMS_0  "ALARM System alarms" %
%   N10:7  SYSTEM_ALARMS_1  "ALARM System alarms" %
%   N10:11  SYSTEM_ALARMS_2 %
%   N16:6/0  ADS_A_HT_PURIFY_ALM  "ALARM ADS A Purify High Temp" %
%   N17:6/0  ADS_B_HT_PURIFY_ALM  "ALARM ADS B Purify High Temp" %
%   B26:20  GETTER_ALARMS %
%   B26:22/5  OPEN_TC5_ALARM %
%   N10:6/6  OPEN_TC6_ALARM %
%   N10:16/0  ACTIVE_SYSTEM_ALARM %

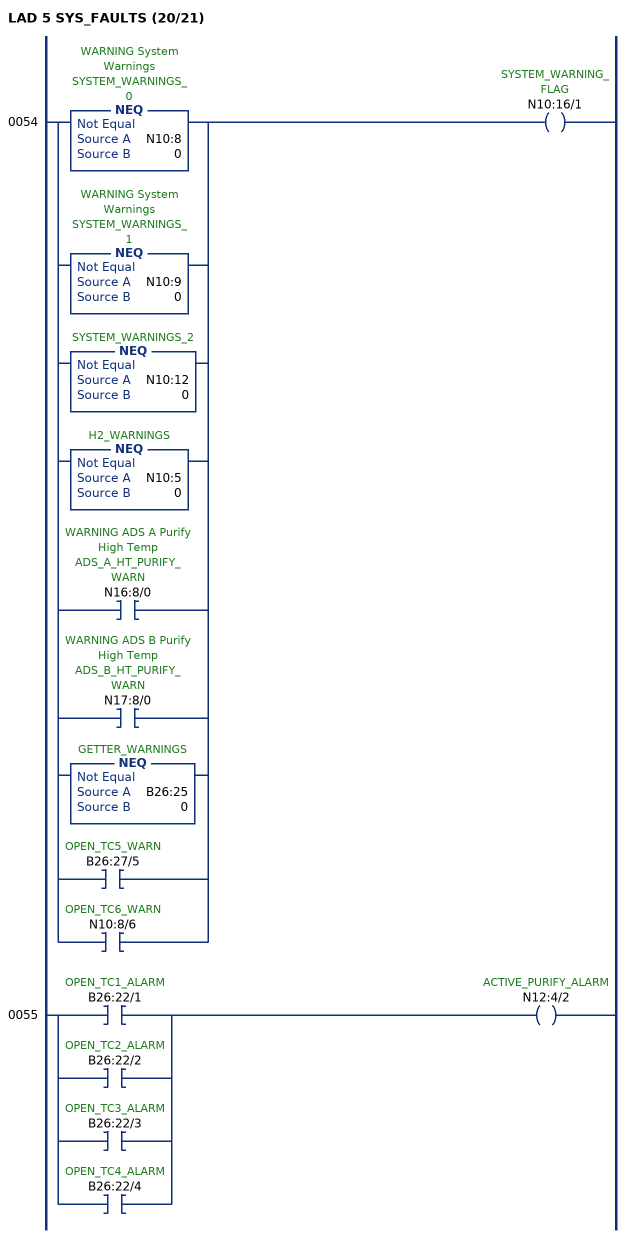
% Rung: 54 %
SOR BST NEQ N10:8 0 NXB NEQ N10:9 0 NXB NEQ N10:12 0 NXB NEQ N10:5 0 NXB XIC N16:8/0 NXB XIC N17:8/0 NXB NEQ B26:25 0 NXB XIC B26:27/5 NXB XIC N10:8/6 BND OTE N10:16/1 EOR
%   N10:8  SYSTEM_WARNINGS_0  "WARNING System Warnings" %
%   N10:9  SYSTEM_WARNINGS_1  "WARNING System Warnings" %
%   N10:12  SYSTEM_WARNINGS_2 %
%   N10:5  H2_WARNINGS %
%   N16:8/0  ADS_A_HT_PURIFY_WARN  "WARNING ADS A Purify High Temp" %
%   N17:8/0  ADS_B_HT_PURIFY_WARN  "WARNING ADS B Purify High Temp" %
%   B26:25  GETTER_WARNINGS %
%   B26:27/5  OPEN_TC5_WARN %
%   N10:8/6  OPEN_TC6_WARN %
%   N10:16/1  SYSTEM_WARNING_FLAG %
% Rung: 55 %
SOR BST XIC B26:22/1 NXB XIC B26:22/2 NXB XIC B26:22/3 NXB XIC B26:22/4 BND OTE N12:4/2 EOR
%   B26:22/1  OPEN_TC1_ALARM %
%   B26:22/2  OPEN_TC2_ALARM %
%   B26:22/3  OPEN_TC3_ALARM %
%   B26:22/4  OPEN_TC4_ALARM %
%   N12:4/2  ACTIVE_PURIFY_ALARM %

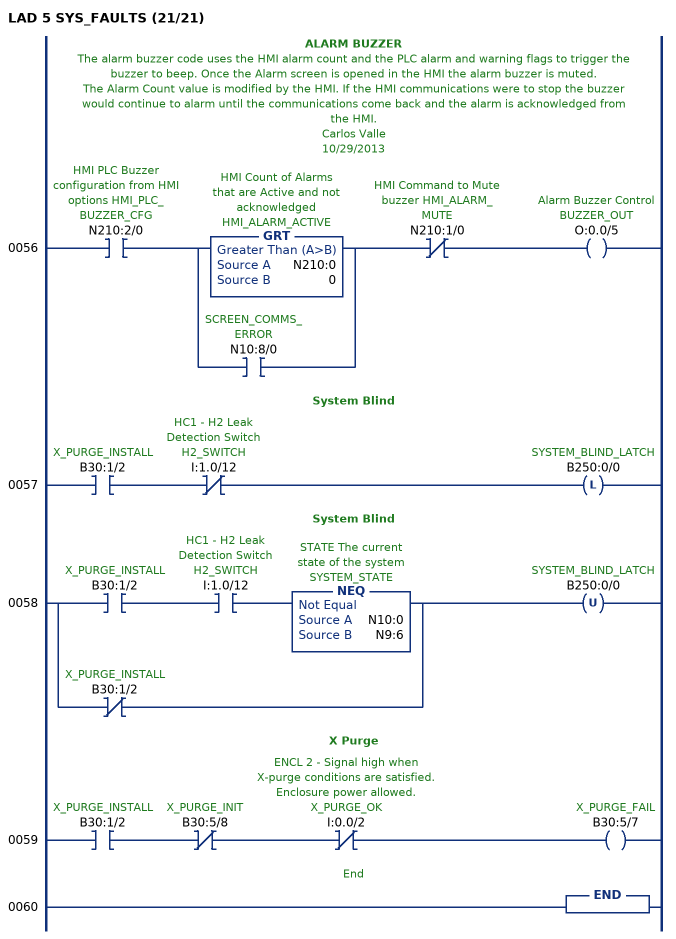
% Rung: 56 %
% TITLE: ALARM BUZZER %
% The alarm buzzer code uses the HMI alarm count and the PLC alarm and warning flags to trigger the buzzer to beep. Once the Alarm screen is opened in the HMI the alarm buzzer is muted.
% The Alarm Count value is modified by the HMI. If the HMI communications were to stop the buzzer would continue to alarm until the communications come back and the alarm is acknowledged from the HMI.
% Carlos Valle
% 10/29/2013 %
SOR XIC N210:2/0 BST GRT N210:0 0 NXB XIC N10:8/0 BND XIO N210:1/0 OTE O:0.0/5 EOR
%   N210:2/0  HMI_PLC_BUZZER_CFG  "HMI PLC Buzzer configuration from HMI options" %
%   N210:0  HMI_ALARM_ACTIVE  "HMI Count of Alarms that are Active and not acknowledged" %
%   N10:8/0  SCREEN_COMMS_ERROR %
%   N210:1/0  HMI_ALARM_MUTE  "HMI Command to Mute buzzer" %
%   O:0.0/5  BUZZER_OUT  "Alarm Buzzer Control" %
% Rung: 57 %
% TITLE: System Blind %
SOR XIC B30:1/2 XIO I:1.0/12 OTL B250:0/0 EOR
%   B30:1/2  X_PURGE_INSTALL %
%   I:1.0/12  H2_SWITCH  "HC1 - H2 Leak Detection Switch" %
%   B250:0/0  SYSTEM_BLIND_LATCH %
% Rung: 58 %
% TITLE: System Blind %
SOR BST XIC B30:1/2 XIC I:1.0/12 NEQ N10:0 N9:6 NXB XIO B30:1/2 BND OTU B250:0/0 EOR
%   B30:1/2  X_PURGE_INSTALL %
%   I:1.0/12  H2_SWITCH  "HC1 - H2 Leak Detection Switch" %
%   N10:0  SYSTEM_STATE  "STATE The current state of the system" %
%   N9:6  SYSTEM_PURGE %
%   B250:0/0  SYSTEM_BLIND_LATCH %
% Rung: 59 %
% TITLE: X Purge %
SOR XIC B30:1/2 XIO B30:5/8 XIO I:0.0/2 OTE B30:5/7 EOR
%   B30:1/2  X_PURGE_INSTALL %
%   B30:5/8  X_PURGE_INIT %
%   I:0.0/2  X_PURGE_OK  "ENCL 2 - Signal high when X-purge conditions are satisfied. Enclosure power allowed." %
%   B30:5/7  X_PURGE_FAIL %
% Rung: 60 %
% End %
SOR END EOR

LADDER 6 "SYSTEM"    % Controls the system %
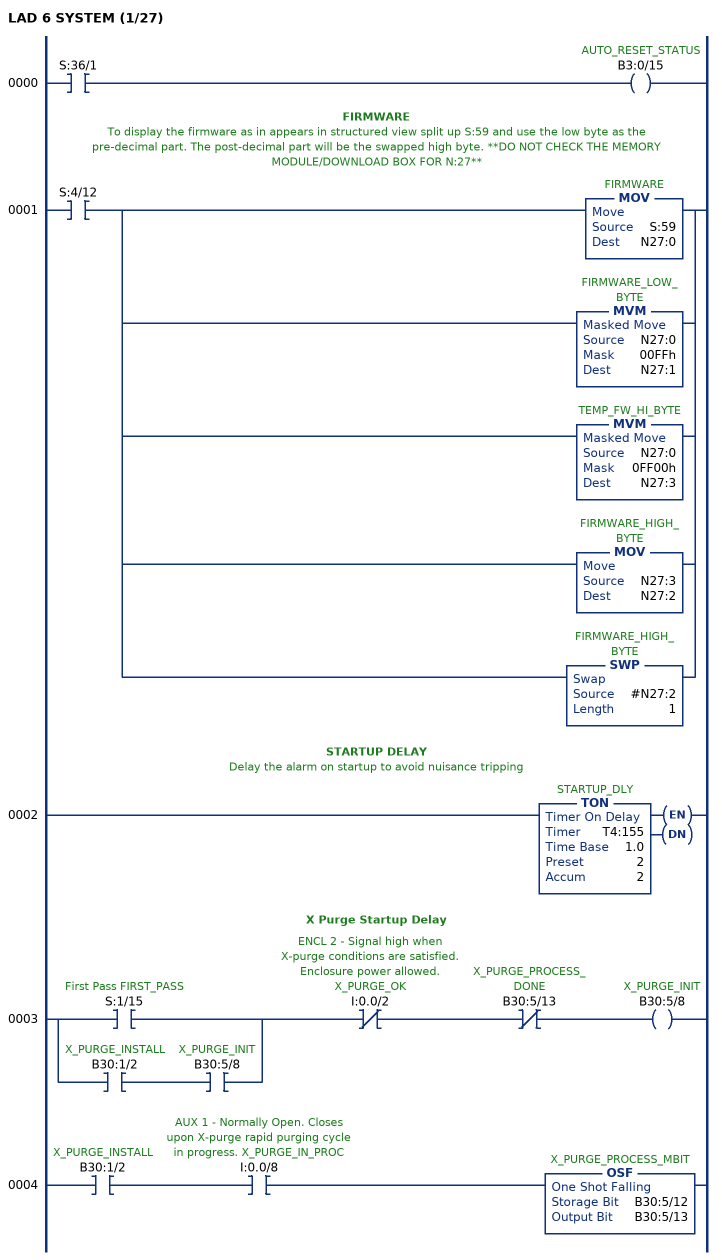
% Rung: 0 %
SOR XIC S:36/1 OTE B3:0/15 EOR
%   B3:0/15  AUTO_RESET_STATUS %
% Rung: 1 %
% TITLE: FIRMWARE %
% To display the firmware as in appears in structured view split up S:59 and use the low byte as the pre-decimal part. The post-decimal part will be the swapped high byte. **DO NOT CHECK THE MEMORY MODULE/DOWNLOAD BOX FOR N:27** %
SOR XIC S:4/12 BST MOV S:59 N27:0 NXB MVM N27:0 00FFh N27:1 NXB MVM N27:0 0FF00h N27:3 NXB MOV N27:3 N27:2 NXB SWP #N27:2 1 BND EOR
%   S:59  "Operating System FRN" %
%   N27:0  FIRMWARE %
%   N27:1  FIRMWARE_LOW_BYTE %
%   N27:3  TEMP_FW_HI_BYTE %
%   N27:2  FIRMWARE_HIGH_BYTE %
% Rung: 2 %
% TITLE: STARTUP DELAY %
% Delay the alarm on startup to avoid nuisance tripping %
SOR TON T4:155 1.0 2 2 EOR
%   T4:155  STARTUP_DLY %
% Rung: 3 %
% TITLE: X Purge Startup Delay %
SOR BST XIC S:1/15 NXB XIC B30:1/2 XIC B30:5/8 BND XIO I:0.0/2 XIO B30:5/13 OTE B30:5/8 EOR
%   S:1/15  FIRST_PASS  "First Pass" %
%   B30:1/2  X_PURGE_INSTALL %
%   B30:5/8  X_PURGE_INIT %
%   I:0.0/2  X_PURGE_OK  "ENCL 2 - Signal high when X-purge conditions are satisfied. Enclosure power allowed." %
%   B30:5/13  X_PURGE_PROCESS_DONE %
% Rung: 4 %
SOR XIC B30:1/2 XIC I:0.0/8 OSF B30:5/12 B30:5/13 EOR
%   B30:1/2  X_PURGE_INSTALL %
%   I:0.0/8  X_PURGE_IN_PROC  "AUX 1 - Normally Open. Closes upon X-purge rapid purging cycle in progress." %
%   B30:5/12  X_PURGE_PROCESS_MBIT %
%   B30:5/13  X_PURGE_PROCESS_DONE %

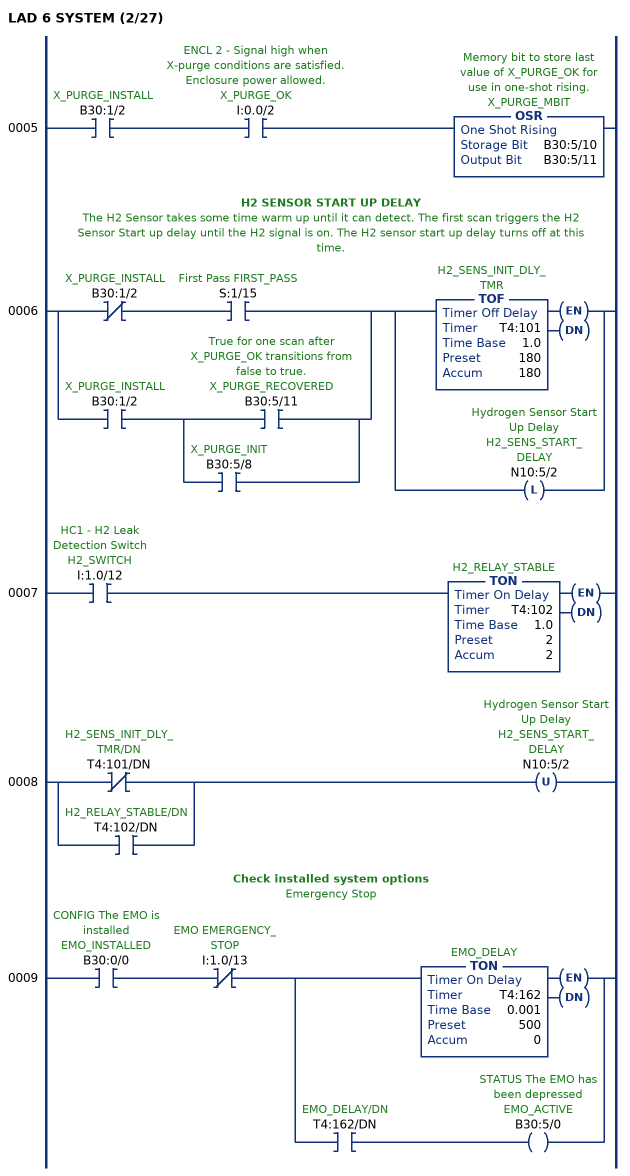
% Rung: 5 %
SOR XIC B30:1/2 XIC I:0.0/2 OSR B30:5/10 B30:5/11 EOR
%   B30:1/2  X_PURGE_INSTALL %
%   I:0.0/2  X_PURGE_OK  "ENCL 2 - Signal high when X-purge conditions are satisfied. Enclosure power allowed." %
%   B30:5/10  X_PURGE_MBIT  "Memory bit to store last value of X_PURGE_OK for use in one-shot rising." %
%   B30:5/11  X_PURGE_RECOVERED  "True for one scan after X_PURGE_OK transitions from false to true." %
% Rung: 6 %
% TITLE: H2 SENSOR START UP DELAY %
% The H2 Sensor takes some time warm up until it can detect. The first scan triggers the H2 Sensor Start up delay until the H2 signal is on. The H2 sensor start up delay turns off at this time. %
SOR BST XIO B30:1/2 XIC S:1/15 NXB XIC B30:1/2 BST XIC B30:5/11 NXB XIC B30:5/8 BND BND BST TOF T4:101 1.0 180 180 NXB OTL N10:5/2 BND EOR
%   B30:1/2  X_PURGE_INSTALL %
%   S:1/15  FIRST_PASS  "First Pass" %
%   B30:5/11  X_PURGE_RECOVERED  "True for one scan after X_PURGE_OK transitions from false to true." %
%   B30:5/8  X_PURGE_INIT %
%   T4:101  H2_SENS_INIT_DLY_TMR %
%   N10:5/2  H2_SENS_START_DELAY  "Hydrogen Sensor Start Up Delay" %
% Rung: 7 %
SOR XIC I:1.0/12 TON T4:102 1.0 2 2 EOR
%   I:1.0/12  H2_SWITCH  "HC1 - H2 Leak Detection Switch" %
%   T4:102  H2_RELAY_STABLE %
% Rung: 8 %
SOR BST XIO T4:101/DN NXB XIC T4:102/DN BND OTU N10:5/2 EOR
%   T4:101  H2_SENS_INIT_DLY_TMR %
%   T4:102  H2_RELAY_STABLE %
%   N10:5/2  H2_SENS_START_DELAY  "Hydrogen Sensor Start Up Delay" %
% Rung: 9 %
% TITLE: Check installed system options %
% Emergency Stop %
SOR XIC B30:0/0 XIO I:1.0/13 BST TON T4:162 0.001 500 0 NXB XIC T4:162/DN OTE B30:5/0 BND EOR
%   B30:0/0  EMO_INSTALLED  "CONFIG The EMO is installed" %
%   I:1.0/13  EMERGENCY_STOP  "EMO" %
%   T4:162  EMO_DELAY %
%   B30:5/0  EMO_ACTIVE  "STATUS The EMO has been depressed" %

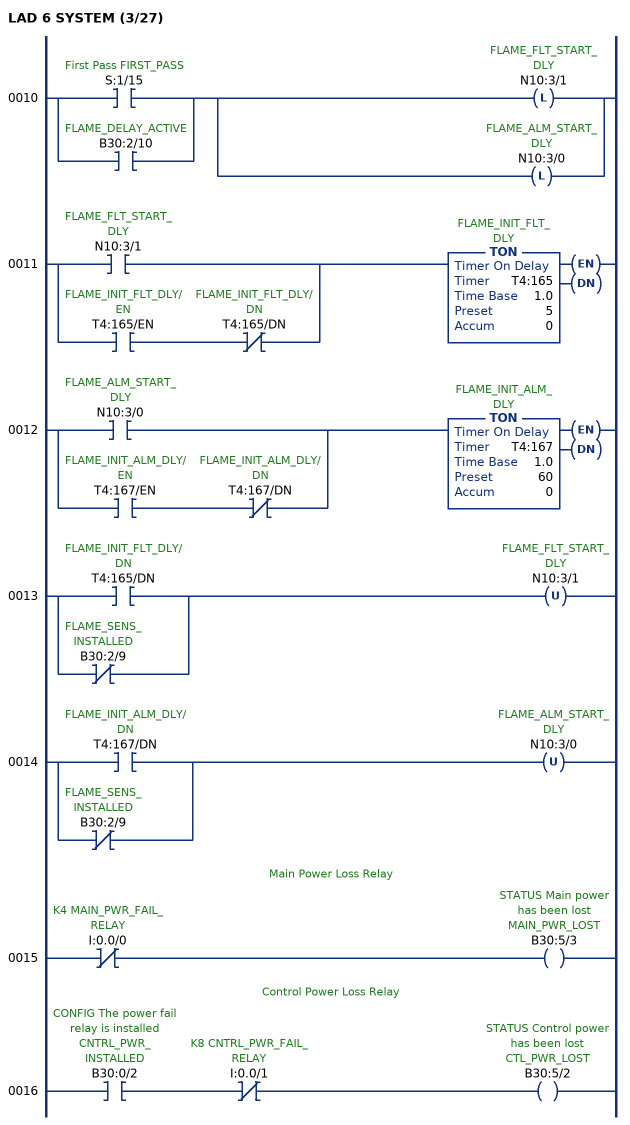
% Rung: 10 %
SOR BST XIC S:1/15 NXB XIC B30:2/10 BND BST OTL N10:3/1 NXB OTL N10:3/0 BND EOR
%   S:1/15  FIRST_PASS  "First Pass" %
%   B30:2/10  FLAME_DELAY_ACTIVE %
%   N10:3/1  FLAME_FLT_START_DLY %
%   N10:3/0  FLAME_ALM_START_DLY %
% Rung: 11 %
SOR BST XIC N10:3/1 NXB XIC T4:165/EN XIO T4:165/DN BND TON T4:165 1.0 5 0 EOR
%   N10:3/1  FLAME_FLT_START_DLY %
%   T4:165  FLAME_INIT_FLT_DLY %
% Rung: 12 %
SOR BST XIC N10:3/0 NXB XIC T4:167/EN XIO T4:167/DN BND TON T4:167 1.0 60 0 EOR
%   N10:3/0  FLAME_ALM_START_DLY %
%   T4:167  FLAME_INIT_ALM_DLY %
% Rung: 13 %
SOR BST XIC T4:165/DN NXB XIO B30:2/9 BND OTU N10:3/1 EOR
%   T4:165  FLAME_INIT_FLT_DLY %
%   B30:2/9  FLAME_SENS_INSTALLED %
%   N10:3/1  FLAME_FLT_START_DLY %
% Rung: 14 %
SOR BST XIC T4:167/DN NXB XIO B30:2/9 BND OTU N10:3/0 EOR
%   T4:167  FLAME_INIT_ALM_DLY %
%   B30:2/9  FLAME_SENS_INSTALLED %
%   N10:3/0  FLAME_ALM_START_DLY %
% Rung: 15 %
% Main Power Loss Relay %
SOR XIO I:0.0/0 OTE B30:5/3 EOR
%   I:0.0/0  MAIN_PWR_FAIL_RELAY  "K4" %
%   B30:5/3  MAIN_PWR_LOST  "STATUS Main power has been lost" %
% Rung: 16 %
% Control Power Loss Relay %
SOR XIC B30:0/2 XIO I:0.0/1 OTE B30:5/2 EOR
%   B30:0/2  CNTRL_PWR_INSTALLED  "CONFIG The power fail relay is installed" %
%   I:0.0/1  CNTRL_PWR_FAIL_RELAY  "K8" %
%   B30:5/2  CTL_PWR_LOST  "STATUS Control power has been lost" %

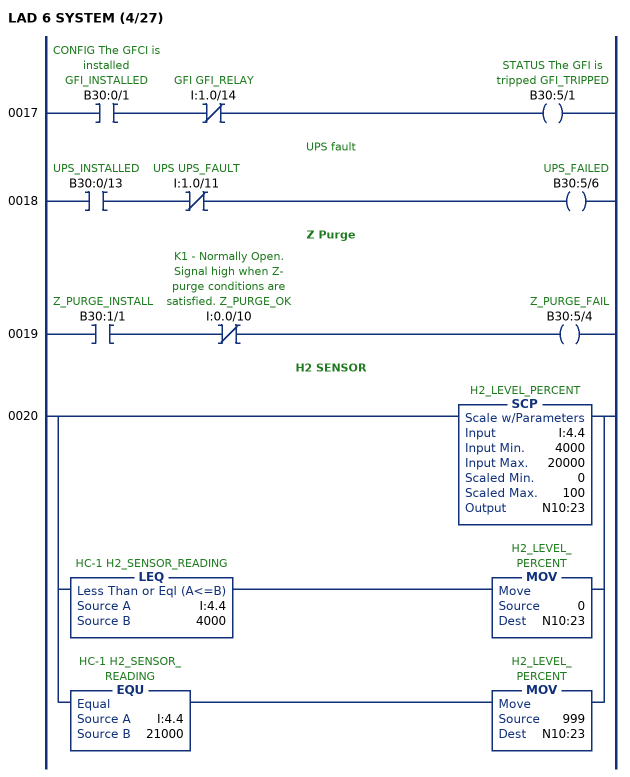
% Rung: 17 %
SOR XIC B30:0/1 XIO I:1.0/14 OTE B30:5/1 EOR
%   B30:0/1  GFI_INSTALLED  "CONFIG The GFCI is installed" %
%   I:1.0/14  GFI_RELAY  "GFI" %
%   B30:5/1  GFI_TRIPPED  "STATUS The GFI is tripped" %
% Rung: 18 %
% UPS fault %
SOR XIC B30:0/13 XIO I:1.0/11 OTE B30:5/6 EOR
%   B30:0/13  UPS_INSTALLED %
%   I:1.0/11  UPS_FAULT  "UPS" %
%   B30:5/6  UPS_FAILED %
% Rung: 19 %
% TITLE: Z Purge %
SOR XIC B30:1/1 XIO I:0.0/10 OTE B30:5/4 EOR
%   B30:1/1  Z_PURGE_INSTALL %
%   I:0.0/10  Z_PURGE_OK  "K1 - Normally Open. Signal high when Z- purge conditions are satisfied." %
%   B30:5/4  Z_PURGE_FAIL %
% Rung: 20 %
% TITLE: H2 SENSOR %
SOR BST SCP I:4.4 4000 20000 0 100 N10:23 NXB LEQ I:4.4 4000 MOV 0 N10:23 NXB EQU I:4.4 21000 MOV 999 N10:23 BND EOR
%   I:4.4  H2_SENSOR_READING  "HC-1" %
%   N10:23  H2_LEVEL_PERCENT %

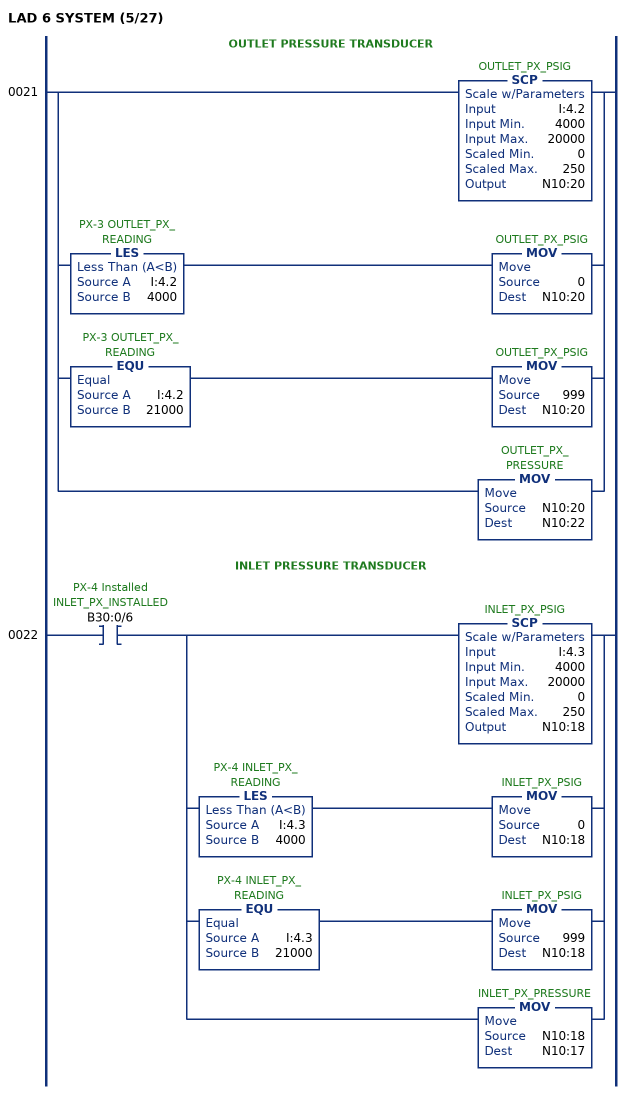
% Rung: 21 %
% TITLE: OUTLET PRESSURE TRANSDUCER %
SOR BST SCP I:4.2 4000 20000 0 250 N10:20 NXB LES I:4.2 4000 MOV 0 N10:20 NXB EQU I:4.2 21000 MOV 999 N10:20 NXB MOV N10:20 N10:22 BND EOR
%   I:4.2  OUTLET_PX_READING  "PX-3" %
%   N10:20  OUTLET_PX_PSIG %
%   N10:22  OUTLET_PX_PRESSURE %
% Rung: 22 %
% TITLE: INLET PRESSURE TRANSDUCER %
SOR XIC B30:0/6 BST SCP I:4.3 4000 20000 0 250 N10:18 NXB LES I:4.3 4000 MOV 0 N10:18 NXB EQU I:4.3 21000 MOV 999 N10:18 NXB MOV N10:18 N10:17 BND EOR
%   B30:0/6  INLET_PX_INSTALLED  "PX-4 Installed" %
%   I:4.3  INLET_PX_READING  "PX-4" %
%   N10:18  INLET_PX_PSIG %
%   N10:17  INLET_PX_PRESSURE %

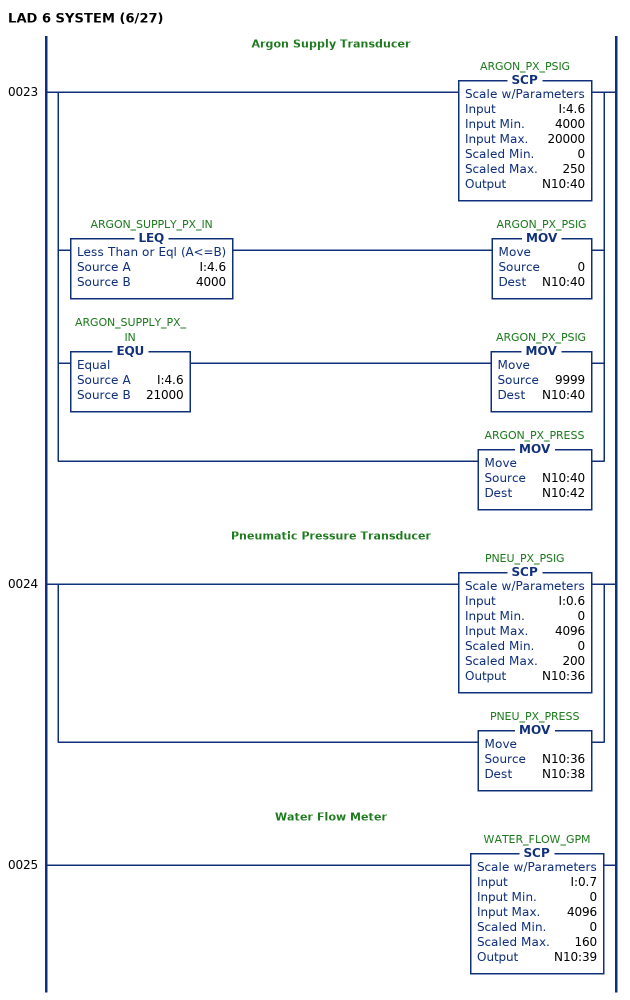
% Rung: 23 %
% TITLE: Argon Supply Transducer %
SOR BST SCP I:4.6 4000 20000 0 250 N10:40 NXB LEQ I:4.6 4000 MOV 0 N10:40 NXB EQU I:4.6 21000 MOV 9999 N10:40 NXB MOV N10:40 N10:42 BND EOR
%   I:4.6  ARGON_SUPPLY_PX_IN %
%   N10:40  ARGON_PX_PSIG %
%   N10:42  ARGON_PX_PRESS %
% Rung: 24 %
% TITLE: Pneumatic Pressure Transducer %
SOR BST SCP I:0.6 0 4096 0 200 N10:36 NXB MOV N10:36 N10:38 BND EOR
%   I:0.6  PNEU_PX_IN  "PX5" %
%   N10:36  PNEU_PX_PSIG %
%   N10:38  PNEU_PX_PRESS %
% Rung: 25 %
% TITLE: Water Flow Meter %
SOR SCP I:0.7 0 4096 0 160 N10:39 EOR
%   I:0.7  WATER_FLOW_IN %
%   N10:39  WATER_FLOW_GPM %

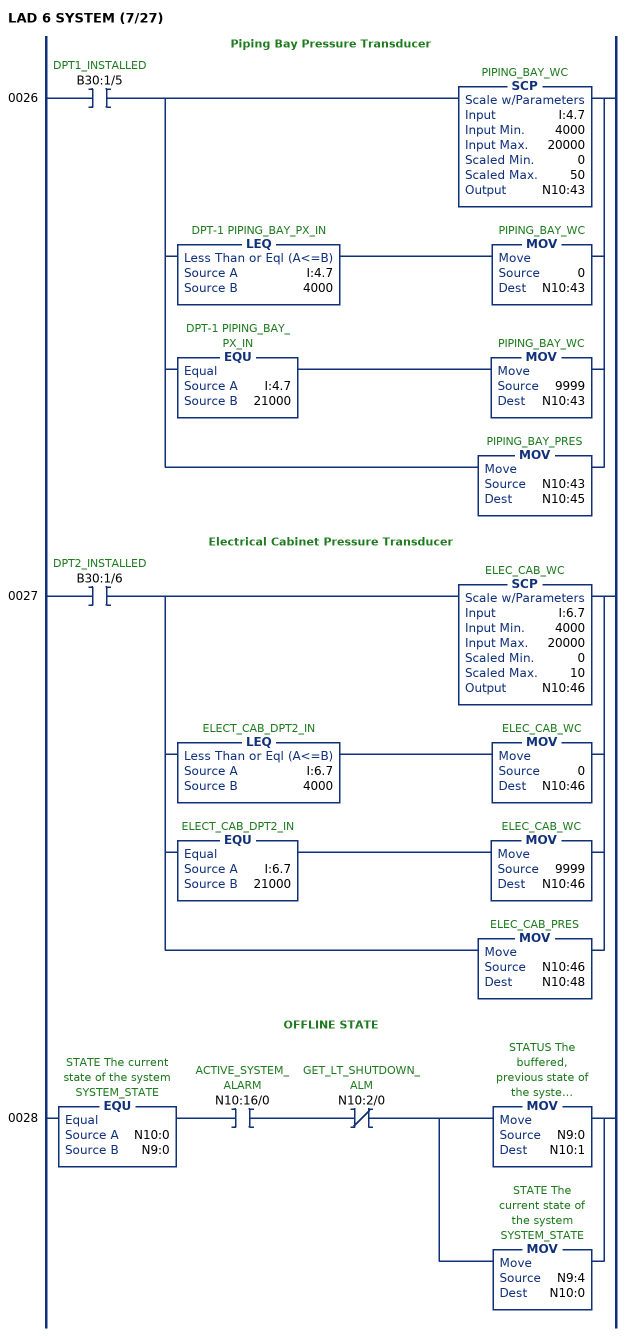
% Rung: 26 %
% TITLE: Piping Bay Pressure Transducer %
SOR XIC B30:1/5 BST SCP I:4.7 4000 20000 0 50 N10:43 NXB LEQ I:4.7 4000 MOV 0 N10:43 NXB EQU I:4.7 21000 MOV 9999 N10:43 NXB MOV N10:43 N10:45 BND EOR
%   B30:1/5  DPT1_INSTALLED %
%   I:4.7  PIPING_BAY_PX_IN  "DPT-1" %
%   N10:43  PIPING_BAY_WC %
%   N10:45  PIPING_BAY_PRES %
% Rung: 27 %
% TITLE: Electrical Cabinet Pressure Transducer %
SOR XIC B30:1/6 BST SCP I:6.7 4000 20000 0 10 N10:46 NXB LEQ I:6.7 4000 MOV 0 N10:46 NXB EQU I:6.7 21000 MOV 9999 N10:46 NXB MOV N10:46 N10:48 BND EOR
%   B30:1/6  DPT2_INSTALLED %
%   I:6.7  ELECT_CAB_DPT2_IN %
%   N10:46  ELEC_CAB_WC %
%   N10:48  ELEC_CAB_PRES %
% Rung: 28 %
% TITLE: OFFLINE STATE %
SOR EQU N10:0 N9:0 XIC N10:16/0 XIO N10:2/0 BST MOV N9:0 N10:1 NXB MOV N9:4 N10:0 BND EOR
%   N10:0  SYSTEM_STATE  "STATE The current state of the system" %
%   N9:0  SYSTEM_OFFLINE %
%   N10:16/0  ACTIVE_SYSTEM_ALARM %
%   N10:2/0  GET_LT_SHUTDOWN_ALM %
%   N10:1  SYSTEM_STATE_BUFFER  "STATUS The buffered, previous state of the system" %
%   N9:4  SYSTEM_ALARM  "STATE System Alarm" %

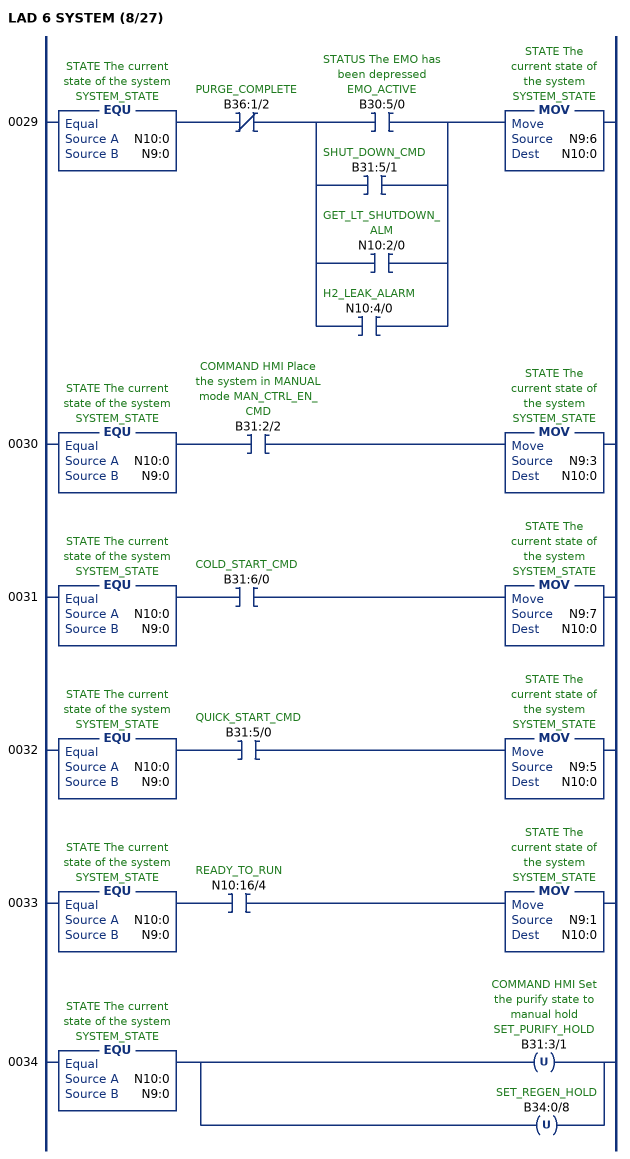
% Rung: 29 %
SOR EQU N10:0 N9:0 XIO B36:1/2 BST XIC B30:5/0 NXB XIC B31:5/1 NXB XIC N10:2/0 NXB XIC N10:4/0 BND MOV N9:6 N10:0 EOR
%   N10:0  SYSTEM_STATE  "STATE The current state of the system" %
%   N9:0  SYSTEM_OFFLINE %
%   B36:1/2  PURGE_COMPLETE %
%   B30:5/0  EMO_ACTIVE  "STATUS The EMO has been depressed" %
%   B31:5/1  SHUT_DOWN_CMD %
%   N10:2/0  GET_LT_SHUTDOWN_ALM %
%   N10:4/0  H2_LEAK_ALARM %
%   N9:6  SYSTEM_PURGE %
% Rung: 30 %
SOR EQU N10:0 N9:0 XIC B31:2/2 MOV N9:3 N10:0 EOR
%   N10:0  SYSTEM_STATE  "STATE The current state of the system" %
%   N9:0  SYSTEM_OFFLINE %
%   B31:2/2  MAN_CTRL_EN_CMD  "COMMAND HMI Place the system in MANUAL mode" %
%   N9:3  SYSTEM_MANUAL  "STATE System Manual" %
% Rung: 31 %
SOR EQU N10:0 N9:0 XIC B31:6/0 MOV N9:7 N10:0 EOR
%   N10:0  SYSTEM_STATE  "STATE The current state of the system" %
%   N9:0  SYSTEM_OFFLINE %
%   B31:6/0  COLD_START_CMD %
%   N9:7  SYSTEM_COLD_START %
% Rung: 32 %
SOR EQU N10:0 N9:0 XIC B31:5/0 MOV N9:5 N10:0 EOR
%   N10:0  SYSTEM_STATE  "STATE The current state of the system" %
%   N9:0  SYSTEM_OFFLINE %
%   B31:5/0  QUICK_START_CMD %
%   N9:5  SYSTEM_QUICK_START %
% Rung: 33 %
SOR EQU N10:0 N9:0 XIC N10:16/4 MOV N9:1 N10:0 EOR
%   N10:0  SYSTEM_STATE  "STATE The current state of the system" %
%   N9:0  SYSTEM_OFFLINE %
%   N10:16/4  READY_TO_RUN %
%   N9:1  SYSTEM_STANDBY  "STATE System Process" %
% Rung: 34 %
SOR EQU N10:0 N9:0 BST OTU B31:3/1 NXB OTU B34:0/8 BND EOR
%   N10:0  SYSTEM_STATE  "STATE The current state of the system" %
%   N9:0  SYSTEM_OFFLINE %
%   B31:3/1  SET_PURIFY_HOLD  "COMMAND HMI Set the purify state to manual hold" %
%   B34:0/8  SET_REGEN_HOLD %

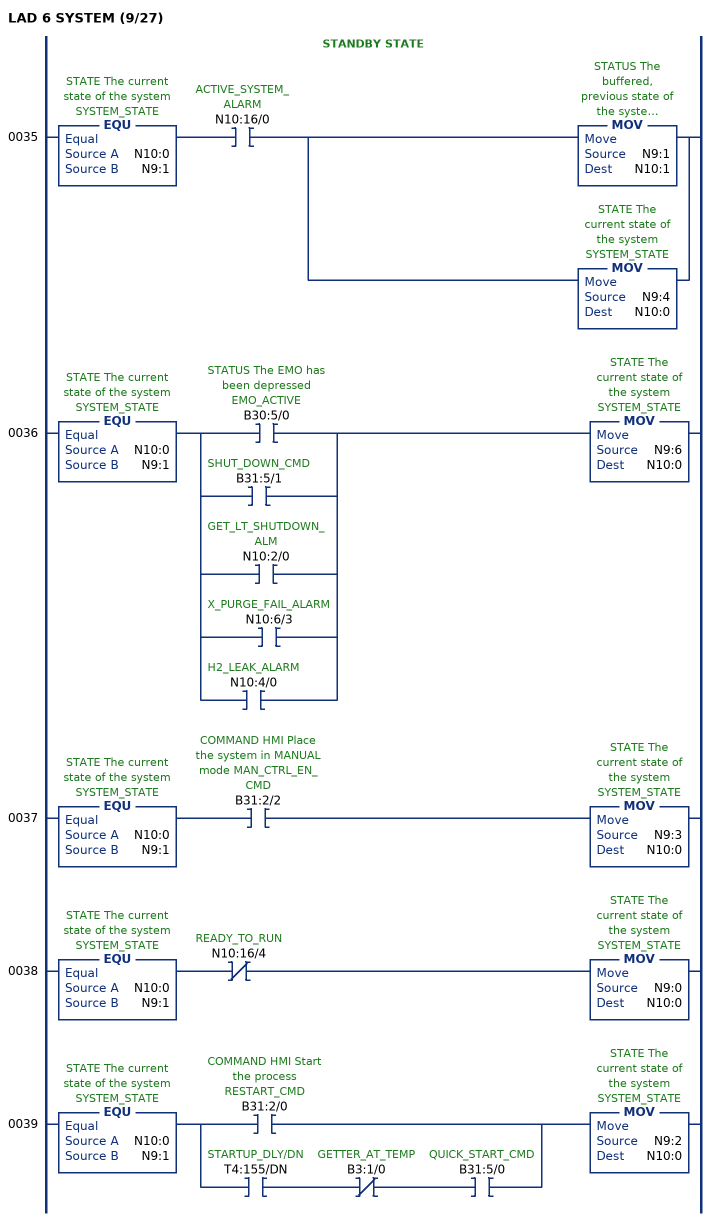
% Rung: 35 %
% TITLE: STANDBY STATE %
SOR EQU N10:0 N9:1 XIC N10:16/0 BST MOV N9:1 N10:1 NXB MOV N9:4 N10:0 BND EOR
%   N10:0  SYSTEM_STATE  "STATE The current state of the system" %
%   N9:1  SYSTEM_STANDBY  "STATE System Process" %
%   N10:16/0  ACTIVE_SYSTEM_ALARM %
%   N10:1  SYSTEM_STATE_BUFFER  "STATUS The buffered, previous state of the system" %
%   N9:4  SYSTEM_ALARM  "STATE System Alarm" %
% Rung: 36 %
SOR EQU N10:0 N9:1 BST XIC B30:5/0 NXB XIC B31:5/1 NXB XIC N10:2/0 NXB XIC N10:6/3 NXB XIC N10:4/0 BND MOV N9:6 N10:0 EOR
%   N10:0  SYSTEM_STATE  "STATE The current state of the system" %
%   N9:1  SYSTEM_STANDBY  "STATE System Process" %
%   B30:5/0  EMO_ACTIVE  "STATUS The EMO has been depressed" %
%   B31:5/1  SHUT_DOWN_CMD %
%   N10:2/0  GET_LT_SHUTDOWN_ALM %
%   N10:6/3  X_PURGE_FAIL_ALARM %
%   N10:4/0  H2_LEAK_ALARM %
%   N9:6  SYSTEM_PURGE %
% Rung: 37 %
SOR EQU N10:0 N9:1 XIC B31:2/2 MOV N9:3 N10:0 EOR
%   N10:0  SYSTEM_STATE  "STATE The current state of the system" %
%   N9:1  SYSTEM_STANDBY  "STATE System Process" %
%   B31:2/2  MAN_CTRL_EN_CMD  "COMMAND HMI Place the system in MANUAL mode" %
%   N9:3  SYSTEM_MANUAL  "STATE System Manual" %
% Rung: 38 %
SOR EQU N10:0 N9:1 XIO N10:16/4 MOV N9:0 N10:0 EOR
%   N10:0  SYSTEM_STATE  "STATE The current state of the system" %
%   N9:1  SYSTEM_STANDBY  "STATE System Process" %
%   N10:16/4  READY_TO_RUN %
%   N9:0  SYSTEM_OFFLINE %
% Rung: 39 %
SOR EQU N10:0 N9:1 BST XIC B31:2/0 NXB XIC T4:155/DN XIO B3:1/0 XIC B31:5/0 BND MOV N9:2 N10:0 EOR
%   N10:0  SYSTEM_STATE  "STATE The current state of the system" %
%   N9:1  SYSTEM_STANDBY  "STATE System Process" %
%   B31:2/0  RESTART_CMD  "COMMAND HMI Start the process" %
%   T4:155  STARTUP_DLY %
%   B3:1/0  GETTER_AT_TEMP %
%   B31:5/0  QUICK_START_CMD %
%   N9:2  SYSTEM_PROCESS  "STATE System Process" %

